LIN {X 50.071,Y -41.479,Z -55.435,A -90.000,B 90.000,C 0.000} C_DIS
LIN {X 50.212,Y -41.479,Z -55.447,A -90.000,B 90.000,C 0.000} C_DIS
LIN {X 50.447,Y -41.466,Z -55.476,A -90.000,B 90.000,C 0.000} C_DIS
LIN {X 50.555,Y -41.461,Z -55.492,A -90.000,B 90.000,C 0.000} C_DIS
LIN {X 50.778,Y -41.444,Z -55.543,A -90.000,B 90.000,C 0.000} C_DIS
LIN {X 51.194,Y -41.423,Z -55.655,A -90.000,B 90.000,C 0.000} C_DIS
LIN {X 51.382,Y -41.418,Z -55.709,A -90.000,B 90.000,C 0.000} C_DIS
LIN {X 51.626,Y -41.420,Z -55.793,A -90.000,B 90.000,C 0.000} C_DIS
LIN {X 51.729,Y -41.422,Z -55.832,A -90.000,B 90.000,C 0.000} C_DIS
LIN {X 52.257,Y -41.443,Z -56.046,A -90.000,B 90.000,C 0.000} C_DIS
LIN {X 52.585,Y -41.450,Z -56.183,A -90.000,B 90.000,C 0.000} C_DIS
LIN {X 52.911,Y -41.433,Z -56.335,A -90.000,B 90.000,C 0.000} C_DIS
LIN {X 53.221,Y -41.399,Z -56.488,A -90.000,B 90.000,C 0.000} C_DIS
LIN {X 53.268,Y -41.394,Z -56.511,A -90.000,B 90.000,C 0.000} C_DIS
LIN {X 53.605,Y -41.331,Z -56.691,A -90.000,B 90.000,C 0.000} C_DIS
LIN {X 53.739,Y -41.308,Z -56.767,A -90.000,B 90.000,C 0.000} C_DIS
LIN {X 53.739,Y -60.000,Z -56.767,A -90.000,B 90.000,C 0.000} C_DIS
LIN {X 39.737,Y -60.000,Z -87.967,A -90.000,B 90.000,C 0.000} C_DIS
LIN {X 39.737,Y -42.859,Z -87.967,A -90.000,B 90.000,C 0.000} C_DIS
LIN {X 40.701,Y -42.857,Z -88.423,A -90.000,B 90.000,C 0.000} C_DIS
LIN {X 40.775,Y -42.860,Z -88.457,A -90.000,B 90.000,C 0.000} C_DIS
LIN {X 41.091,Y -42.861,Z -88.606,A -90.000,B 90.000,C 0.000} C_DIS
LIN {X 41.387,Y -42.856,Z -88.749,A -90.000,B 90.000,C 0.000} C_DIS
LIN {X 41.518,Y -42.856,Z -88.821,A -90.000,B 90.000,C 0.000} C_DIS
LIN {X 41.830,Y -42.856,Z -88.996,A -90.000,B 90.000,C 0.000} C_DIS
LIN {X 41.925,Y -42.857,Z -89.053,A -90.000,B 90.000,C 0.000} C_DIS
LIN {X 42.012,Y -42.859,Z -89.111,A -90.000,B 90.000,C 0.000} C_DIS
LIN {X 42.238,Y -42.866,Z -89.272,A -90.000,B 90.000,C 0.000} C_DIS
LIN {X 42.392,Y -42.871,Z -89.385,A -90.000,B 90.000,C 0.000} C_DIS
LIN {X 42.668,Y -42.871,Z -89.540,A -90.000,B 90.000,C 0.000} C_DIS
LIN {X 43.663,Y -42.840,Z -90.105,A -90.000,B 90.000,C 0.000} C_DIS
LIN {X 43.846,Y -42.837,Z -90.222,A -90.000,B 90.000,C 0.000} C_DIS
LIN {X 44.056,Y -42.836,Z -90.373,A -90.000,B 90.000,C 0.000} C_DIS
LIN {X 44.494,Y -42.834,Z -90.695,A -90.000,B 90.000,C 0.000} C_DIS
LIN {X 44.650,Y -42.831,Z -90.811,A -90.000,B 90.000,C 0.000} C_DIS
LIN {X 44.974,Y -42.816,Z -91.054,A -90.000,B 90.000,C 0.000} C_DIS
LIN {X 45.094,Y -42.815,Z -91.149,A -90.000,B 90.000,C 0.000} C_DIS
LIN {X 45.874,Y -42.815,Z -91.799,A -90.000,B 90.000,C 0.000} C_DIS
LIN {X 45.991,Y -42.817,Z -91.906,A -90.000,B 90.000,C 0.000} C_DIS
LIN {X 46.076,Y -42.820,Z -91.995,A -90.000,B 90.000,C 0.000} C_DIS
LIN {X 46.259,Y -42.829,Z -92.193,A -90.000,B 90.000,C 0.000} C_DIS
LIN {X 46.966,Y -42.829,Z -92.975,A -90.000,B 90.000,C 0.000} C_DIS
LIN {X 47.383,Y -42.820,Z -93.379,A -90.000,B 90.000,C 0.000} C_DIS
LIN {X 47.478,Y -42.813,Z -93.473,A -90.000,B 90.000,C 0.000} C_DIS
LIN {X 47.567,Y -42.807,Z -93.567,A -90.000,B 90.000,C 0.000} C_DIS
LIN {X 47.724,Y -42.799,Z -93.743,A -90.000,B 90.000,C 0.000} C_DIS
LIN {X 47.806,Y -42.796,Z -93.841,A -90.000,B 90.000,C 0.000} C_DIS
LIN {X 48.188,Y -42.784,Z -94.326,A -90.000,B 90.000,C 0.000} C_DIS
LIN {X 48.342,Y -42.784,Z -94.551,A -90.000,B 90.000,C 0.000} C_DIS
LIN {X 48.557,Y -42.792,Z -94.920,A -90.000,B 90.000,C 0.000} C_DIS
LIN {X 49.731,Y -42.798,Z -96.974,A -90.000,B 90.000,C 0.000} C_DIS
LIN {X 50.005,Y -42.776,Z -97.466,A -90.000,B 90.000,C 0.000} C_DIS
LIN {X 50.218,Y -42.754,Z -97.852,A -90.000,B 90.000,C 0.000} C_DIS
LIN {X 50.313,Y -42.746,Z -98.046,A -90.000,B 90.000,C 0.000} C_DIS
LIN {X 50.630,Y -42.732,Z -98.793,A -90.000,B 90.000,C 0.000} C_DIS
LIN {X 50.685,Y -42.731,Z -98.940,A -90.000,B 90.000,C 0.000} C_DIS
LIN {X 50.789,Y -42.732,Z -99.247,A -90.000,B 90.000,C 0.000} C_DIS
LIN {X 50.909,Y -42.728,Z -99.606,A -90.000,B 90.000,C 0.000} C_DIS
LIN {X 50.940,Y -42.728,Z -99.713,A -90.000,B 90.000,C 0.000} C_DIS
LIN {X 51.021,Y -42.724,Z -100.019,A -90.000,B 90.000,C 0.000} C_DIS
LIN {X 51.404,Y -42.715,Z -101.622,A -90.000,B 90.000,C 0.000} C_DIS
LIN {X 51.588,Y -42.705,Z -102.400,A -90.000,B 90.000,C 0.000} C_DIS
LIN {X 51.623,Y -42.698,Z -102.554,A -90.000,B 90.000,C 0.000} C_DIS
LIN {X 51.666,Y -42.691,Z -102.832,A -90.000,B 90.000,C 0.000} C_DIS
LIN {X 51.762,Y -42.691,Z -103.918,A -90.000,B 90.000,C 0.000} C_DIS
LIN {X 51.950,Y -42.585,Z -106.453,A -90.000,B 90.000,C 0.000} C_DIS
LIN {X 51.961,Y -42.579,Z -106.611,A -90.000,B 90.000,C 0.000} C_DIS
LIN {X 51.967,Y -42.576,Z -106.795,A -90.000,B 90.000,C 0.000} C_DIS
LIN {X 51.961,Y -42.576,Z -107.317,A -90.000,B 90.000,C 0.000} C_DIS
LIN {X 51.957,Y -42.578,Z -107.444,A -90.000,B 90.000,C 0.000} C_DIS
LIN {X 51.942,Y -42.583,Z -107.626,A -90.000,B 90.000,C 0.000} C_DIS
LIN {X 51.893,Y -42.599,Z -108.028,A -90.000,B 90.000,C 0.000} C_DIS
LIN {X 51.693,Y -42.585,Z -109.737,A -90.000,B 90.000,C 0.000} C_DIS
LIN {X 51.495,Y -42.558,Z -111.384,A -90.000,B 90.000,C 0.000} C_DIS
LIN {X 51.480,Y -42.556,Z -111.487,A -90.000,B 90.000,C 0.000} C_DIS
LIN {X 51.431,Y -42.553,Z -111.764,A -90.000,B 90.000,C 0.000} C_DIS
LIN {X 51.407,Y -42.554,Z -111.885,A -90.000,B 90.000,C 0.000} C_DIS
LIN {X 51.390,Y -42.555,Z -111.958,A -90.000,B 90.000,C 0.000} C_DIS
LIN {X 51.314,Y -42.552,Z -112.270,A -90.000,B 90.000,C 0.000} C_DIS
LIN {X 51.191,Y -42.541,Z -112.760,A -90.000,B 90.000,C 0.000} C_DIS
LIN {X 50.692,Y -42.505,Z -114.766,A -90.000,B 90.000,C 0.000} C_DIS
LIN {X 50.498,Y -42.486,Z -115.589,A -90.000,B 90.000,C 0.000} C_DIS
LIN {X 50.434,Y -42.486,Z -115.809,A -90.000,B 90.000,C 0.000} C_DIS
LIN {X 50.344,Y -42.494,Z -116.069,A -90.000,B 90.000,C 0.000} C_DIS
LIN {X 49.479,Y -42.446,Z -118.357,A -90.000,B 90.000,C 0.000} C_DIS
LIN {X 49.172,Y -42.430,Z -119.163,A -90.000,B 90.000,C 0.000} C_DIS
LIN {X 49.034,Y -42.425,Z -119.529,A -90.000,B 90.000,C 0.000} C_DIS
LIN {X 48.992,Y -42.424,Z -119.632,A -90.000,B 90.000,C 0.000} C_DIS
LIN {X 48.884,Y -42.426,Z -119.879,A -90.000,B 90.000,C 0.000} C_DIS
LIN {X 48.823,Y -42.428,Z -120.005,A -90.000,B 90.000,C 0.000} C_DIS
LIN {X 48.791,Y -42.431,Z -120.066,A -90.000,B 90.000,C 0.000} C_DIS
LIN {X 48.534,Y -42.422,Z -120.533,A -90.000,B 90.000,C 0.000} C_DIS
LIN {X 47.898,Y -42.413,Z -121.632,A -90.000,B 90.000,C 0.000} C_DIS
LIN {X 46.862,Y -42.389,Z -123.413,A -90.000,B 90.000,C 0.000} C_DIS
LIN {X 46.662,Y -42.391,Z -123.729,A -90.000,B 90.000,C 0.000} C_DIS
LIN {X 46.658,Y -42.391,Z -123.735,A -90.000,B 90.000,C 0.000} C_DIS
LIN {X 46.583,Y -42.387,Z -123.842,A -90.000,B 90.000,C 0.000} C_DIS
LIN {X 46.538,Y -42.386,Z -123.901,A -90.000,B 90.000,C 0.000} C_DIS
LIN {X 46.281,Y -42.383,Z -124.220,A -90.000,B 90.000,C 0.000} C_DIS
LIN {X 44.705,Y -42.346,Z -126.159,A -90.000,B 90.000,C 0.000} C_DIS
LIN {X 43.973,Y -42.339,Z -127.027,A -90.000,B 90.000,C 0.000} C_DIS
LIN {X 43.899,Y -42.333,Z -127.109,A -90.000,B 90.000,C 0.000} C_DIS
LIN {X 43.803,Y -42.329,Z -127.209,A -90.000,B 90.000,C 0.000} C_DIS
LIN {X 41.107,Y -42.265,Z -129.839,A -90.000,B 90.000,C 0.000} C_DIS
LIN {X 40.894,Y -42.262,Z -130.041,A -90.000,B 90.000,C 0.000} C_DIS
LIN {X 40.681,Y -42.253,Z -130.229,A -90.000,B 90.000,C 0.000} C_DIS
LIN {X 38.963,Y -42.211,Z -131.679,A -90.000,B 90.000,C 0.000} C_DIS
LIN {X 37.727,Y -42.184,Z -132.716,A -90.000,B 90.000,C 0.000} C_DIS
LIN {X 37.616,Y -42.182,Z -132.810,A -90.000,B 90.000,C 0.000} C_DIS
LIN {X 37.039,Y -42.183,Z -133.273,A -90.000,B 90.000,C 0.000} C_DIS
LIN {X 34.620,Y -42.128,Z -135.162,A -90.000,B 90.000,C 0.000} C_DIS
LIN {X 33.077,Y -42.091,Z -136.358,A -90.000,B 90.000,C 0.000} C_DIS
LIN {X 32.369,Y -42.096,Z -136.929,A -90.000,B 90.000,C 0.000} C_DIS
LIN {X 31.860,Y -42.079,Z -137.367,A -90.000,B 90.000,C 0.000} C_DIS
LIN {X 31.762,Y -42.078,Z -137.447,A -90.000,B 90.000,C 0.000} C_DIS
LIN {X 30.790,Y -42.057,Z -138.156,A -90.000,B 90.000,C 0.000} C_DIS
LIN {X 30.113,Y -42.060,Z -138.669,A -90.000,B 90.000,C 0.000} C_DIS
LIN {X 28.963,Y -42.027,Z -139.590,A -90.000,B 90.000,C 0.000} C_DIS
LIN {X 28.847,Y -42.027,Z -139.678,A -90.000,B 90.000,C 0.000} C_DIS
LIN {X 28.513,Y -42.013,Z -139.905,A -90.000,B 90.000,C 0.000} C_DIS
LIN {X 27.881,Y -42.005,Z -140.313,A -90.000,B 90.000,C 0.000} C_DIS
LIN {X 26.764,Y -42.006,Z -141.053,A -90.000,B 90.000,C 0.000} C_DIS
LIN {X 25.701,Y -41.985,Z -141.782,A -90.000,B 90.000,C 0.000} C_DIS
LIN {X 25.467,Y -41.978,Z -141.937,A -90.000,B 90.000,C 0.000} C_DIS
LIN {X 25.363,Y -41.981,Z -141.999,A -90.000,B 90.000,C 0.000} C_DIS
LIN {X 25.194,Y -41.978,Z -142.091,A -90.000,B 90.000,C 0.000} C_DIS
LIN {X 23.934,Y -41.975,Z -142.754,A -90.000,B 90.000,C 0.000} C_DIS
LIN {X 22.011,Y -41.953,Z -143.779,A -90.000,B 90.000,C 0.000} C_DIS
LIN {X 21.928,Y -41.954,Z -143.821,A -90.000,B 90.000,C 0.000} C_DIS
LIN {X 21.714,Y -41.959,Z -143.926,A -90.000,B 90.000,C 0.000} C_DIS
LIN {X 21.480,Y -41.961,Z -144.033,A -90.000,B 90.000,C 0.000} C_DIS
LIN {X 21.348,Y -41.966,Z -144.089,A -90.000,B 90.000,C 0.000} C_DIS
LIN {X 18.681,Y -41.946,Z -145.072,A -90.000,B 90.000,C 0.000} C_DIS
LIN {X 17.616,Y -41.939,Z -145.462,A -90.000,B 90.000,C 0.000} C_DIS
LIN {X 17.283,Y -41.941,Z -145.580,A -90.000,B 90.000,C 0.000} C_DIS
LIN {X 16.866,Y -41.961,Z -145.707,A -90.000,B 90.000,C 0.000} C_DIS
LIN {X 16.487,Y -41.974,Z -145.816,A -90.000,B 90.000,C 0.000} C_DIS
LIN {X 14.194,Y -41.972,Z -146.399,A -90.000,B 90.000,C 0.000} C_DIS
LIN {X 12.844,Y -41.974,Z -146.734,A -90.000,B 90.000,C 0.000} C_DIS
LIN {X 12.500,Y -41.983,Z -146.811,A -90.000,B 90.000,C 0.000} C_DIS
LIN {X 12.199,Y -41.993,Z -146.875,A -90.000,B 90.000,C 0.000} C_DIS
LIN {X 11.749,Y -42.015,Z -146.962,A -90.000,B 90.000,C 0.000} C_DIS
LIN {X 11.360,Y -42.023,Z -147.028,A -90.000,B 90.000,C 0.000} C_DIS
LIN {X 9.505,Y -42.021,Z -147.309,A -90.000,B 90.000,C 0.000} C_DIS
LIN {X 7.684,Y -42.033,Z -147.572,A -90.000,B 90.000,C 0.000} C_DIS
LIN {X 7.309,Y -42.042,Z -147.618,A -90.000,B 90.000,C 0.000} C_DIS
LIN {X 7.166,Y -42.049,Z -147.632,A -90.000,B 90.000,C 0.000} C_DIS
LIN {X 6.691,Y -42.078,Z -147.670,A -90.000,B 90.000,C 0.000} C_DIS
LIN {X 6.323,Y -42.091,Z -147.692,A -90.000,B 90.000,C 0.000} C_DIS
LIN {X 5.823,Y -42.090,Z -147.707,A -90.000,B 90.000,C 0.000} C_DIS
LIN {X 3.623,Y -42.092,Z -147.779,A -90.000,B 90.000,C 0.000} C_DIS
LIN {X 3.188,Y -42.091,Z -147.792,A -90.000,B 90.000,C 0.000} C_DIS
LIN {X 2.793,Y -42.094,Z -147.798,A -90.000,B 90.000,C 0.000} C_DIS
LIN {X 2.443,Y -42.104,Z -147.796,A -90.000,B 90.000,C 0.000} C_DIS
LIN {X 2.302,Y -42.111,Z -147.791,A -90.000,B 90.000,C 0.000} C_DIS
LIN {X 2.162,Y -42.121,Z -147.784,A -90.000,B 90.000,C 0.000} C_DIS
LIN {X 1.780,Y -42.138,Z -147.750,A -90.000,B 90.000,C 0.000} C_DIS
LIN {X -1.809,Y -42.140,Z -147.310,A -90.000,B 90.000,C 0.000} C_DIS
LIN {X -2.153,Y -42.146,Z -147.257,A -90.000,B 90.000,C 0.000} C_DIS
LIN {X -2.321,Y -42.149,Z -147.226,A -90.000,B 90.000,C 0.000} C_DIS
LIN {X -2.512,Y -42.161,Z -147.180,A -90.000,B 90.000,C 0.000} C_DIS
LIN {X -5.904,Y -42.185,Z -146.217,A -90.000,B 90.000,C 0.000} C_DIS
LIN {X -6.299,Y -42.185,Z -146.107,A -90.000,B 90.000,C 0.000} C_DIS
LIN {X -6.474,Y -42.187,Z -146.050,A -90.000,B 90.000,C 0.000} C_DIS
LIN {X -6.619,Y -42.192,Z -145.996,A -90.000,B 90.000,C 0.000} C_DIS
LIN {X -6.797,Y -42.187,Z -145.923,A -90.000,B 90.000,C 0.000} C_DIS
LIN {X -6.898,Y -42.187,Z -145.879,A -90.000,B 90.000,C 0.000} C_DIS
LIN {X -9.013,Y -42.202,Z -144.902,A -90.000,B 90.000,C 0.000} C_DIS
LIN {X -10.307,Y -42.229,Z -144.277,A -90.000,B 90.000,C 0.000} C_DIS
LIN {X -10.392,Y -42.227,Z -144.233,A -90.000,B 90.000,C 0.000} C_DIS
LIN {X -10.641,Y -42.224,Z -144.092,A -90.000,B 90.000,C 0.000} C_DIS
LIN {X -10.832,Y -42.222,Z -143.972,A -90.000,B 90.000,C 0.000} C_DIS
LIN {X -10.913,Y -42.223,Z -143.918,A -90.000,B 90.000,C 0.000} C_DIS
LIN {X -11.965,Y -42.251,Z -143.181,A -90.000,B 90.000,C 0.000} C_DIS
LIN {X -13.757,Y -42.332,Z -141.862,A -90.000,B 90.000,C 0.000} C_DIS
LIN {X -13.967,Y -42.332,Z -141.700,A -90.000,B 90.000,C 0.000} C_DIS
LIN {X -14.058,Y -42.333,Z -141.626,A -90.000,B 90.000,C 0.000} C_DIS
LIN {X -14.298,Y -42.335,Z -141.415,A -90.000,B 90.000,C 0.000} C_DIS
LIN {X -14.414,Y -42.339,Z -141.307,A -90.000,B 90.000,C 0.000} C_DIS
LIN {X -14.878,Y -42.372,Z -140.841,A -90.000,B 90.000,C 0.000} C_DIS
LIN {X -15.587,Y -42.405,Z -140.116,A -90.000,B 90.000,C 0.000} C_DIS
LIN {X -15.666,Y -42.411,Z -140.030,A -90.000,B 90.000,C 0.000} C_DIS
LIN {X -15.913,Y -42.435,Z -139.750,A -90.000,B 90.000,C 0.000} C_DIS
LIN {X -16.705,Y -42.506,Z -138.786,A -90.000,B 90.000,C 0.000} C_DIS
LIN {X -16.907,Y -42.509,Z -138.529,A -90.000,B 90.000,C 0.000} C_DIS
LIN {X -17.090,Y -42.502,Z -138.288,A -90.000,B 90.000,C 0.000} C_DIS
LIN {X -17.149,Y -42.500,Z -138.207,A -90.000,B 90.000,C 0.000} C_DIS
LIN {X -17.273,Y -42.500,Z -138.024,A -90.000,B 90.000,C 0.000} C_DIS
LIN {X -17.333,Y -42.502,Z -137.930,A -90.000,B 90.000,C 0.000} C_DIS
LIN {X -17.523,Y -42.510,Z -137.616,A -90.000,B 90.000,C 0.000} C_DIS
LIN {X -17.548,Y -42.512,Z -137.572,A -90.000,B 90.000,C 0.000} C_DIS
LIN {X -18.006,Y -42.548,Z -136.749,A -90.000,B 90.000,C 0.000} C_DIS
LIN {X -18.152,Y -42.554,Z -136.476,A -90.000,B 90.000,C 0.000} C_DIS
LIN {X -18.227,Y -42.560,Z -136.309,A -90.000,B 90.000,C 0.000} C_DIS
LIN {X -18.660,Y -42.596,Z -135.308,A -90.000,B 90.000,C 0.000} C_DIS
LIN {X -18.715,Y -42.603,Z -135.169,A -90.000,B 90.000,C 0.000} C_DIS
LIN {X -18.808,Y -42.619,Z -134.900,A -90.000,B 90.000,C 0.000} C_DIS
LIN {X -18.853,Y -42.629,Z -134.752,A -90.000,B 90.000,C 0.000} C_DIS
LIN {X -18.945,Y -42.658,Z -134.411,A -90.000,B 90.000,C 0.000} C_DIS
LIN {X -19.082,Y -42.685,Z -133.875,A -90.000,B 90.000,C 0.000} C_DIS
LIN {X -19.107,Y -42.689,Z -133.784,A -90.000,B 90.000,C 0.000} C_DIS
LIN {X -19.176,Y -42.693,Z -133.531,A -90.000,B 90.000,C 0.000} C_DIS
LIN {X -19.325,Y -42.693,Z -132.968,A -90.000,B 90.000,C 0.000} C_DIS
LIN {X -19.362,Y -42.695,Z -132.798,A -90.000,B 90.000,C 0.000} C_DIS
LIN {X -19.437,Y -42.713,Z -132.299,A -90.000,B 90.000,C 0.000} C_DIS
LIN {X -19.552,Y -42.713,Z -131.461,A -90.000,B 90.000,C 0.000} C_DIS
LIN {X -19.581,Y -42.717,Z -131.156,A -90.000,B 90.000,C 0.000} C_DIS
LIN {X -19.603,Y -42.724,Z -130.934,A -90.000,B 90.000,C 0.000} C_DIS
LIN {X -19.640,Y -42.751,Z -130.280,A -90.000,B 90.000,C 0.000} C_DIS
LIN {X -19.639,Y -42.759,Z -130.130,A -90.000,B 90.000,C 0.000} C_DIS
LIN {X -19.617,Y -42.789,Z -129.641,A -90.000,B 90.000,C 0.000} C_DIS
LIN {X -19.636,Y -42.801,Z -129.252,A -90.000,B 90.000,C 0.000} C_DIS
LIN {X -19.641,Y -42.803,Z -129.145,A -90.000,B 90.000,C 0.000} C_DIS
LIN {X -19.677,Y -42.803,Z -128.287,A -90.000,B 90.000,C 0.000} C_DIS
LIN {X -19.697,Y -42.805,Z -127.046,A -90.000,B 90.000,C 0.000} C_DIS
LIN {X -19.693,Y -42.809,Z -126.940,A -90.000,B 90.000,C 0.000} C_DIS
LIN {X -19.653,Y -42.844,Z -126.286,A -90.000,B 90.000,C 0.000} C_DIS
LIN {X -19.642,Y -42.858,Z -126.087,A -90.000,B 90.000,C 0.000} C_DIS
LIN {X -19.631,Y -42.879,Z -125.771,A -90.000,B 90.000,C 0.000} C_DIS
LIN {X -19.603,Y -42.899,Z -125.166,A -90.000,B 90.000,C 0.000} C_DIS
LIN {X -19.661,Y -42.899,Z -124.644,A -90.000,B 90.000,C 0.000} C_DIS
LIN {X -19.758,Y -42.891,Z -124.156,A -90.000,B 90.000,C 0.000} C_DIS
LIN {X -19.801,Y -42.891,Z -123.940,A -90.000,B 90.000,C 0.000} C_DIS
LIN {X -20.115,Y -42.903,Z -122.129,A -90.000,B 90.000,C 0.000} C_DIS
LIN {X -20.237,Y -42.923,Z -121.450,A -90.000,B 90.000,C 0.000} C_DIS
LIN {X -20.376,Y -42.942,Z -120.661,A -90.000,B 90.000,C 0.000} C_DIS
LIN {X -20.581,Y -42.942,Z -119.994,A -90.000,B 90.000,C 0.000} C_DIS
LIN {X -21.455,Y -42.935,Z -117.314,A -90.000,B 90.000,C 0.000} C_DIS
LIN {X -21.829,Y -42.941,Z -116.105,A -90.000,B 90.000,C 0.000} C_DIS
LIN {X -22.072,Y -42.942,Z -115.374,A -90.000,B 90.000,C 0.000} C_DIS
LIN {X -22.994,Y -42.949,Z -112.548,A -90.000,B 90.000,C 0.000} C_DIS
LIN {X -23.502,Y -42.948,Z -111.018,A -90.000,B 90.000,C 0.000} C_DIS
LIN {X -23.968,Y -42.918,Z -109.597,A -90.000,B 90.000,C 0.000} C_DIS
LIN {X -23.994,Y -42.917,Z -109.512,A -90.000,B 90.000,C 0.000} C_DIS
LIN {X -24.144,Y -42.910,Z -108.976,A -90.000,B 90.000,C 0.000} C_DIS
LIN {X -24.171,Y -42.910,Z -108.866,A -90.000,B 90.000,C 0.000} C_DIS
LIN {X -24.570,Y -42.910,Z -107.060,A -90.000,B 90.000,C 0.000} C_DIS
LIN {X -24.799,Y -42.909,Z -106.089,A -90.000,B 90.000,C 0.000} C_DIS
LIN {X -24.962,Y -42.917,Z -105.256,A -90.000,B 90.000,C 0.000} C_DIS
LIN {X -25.003,Y -42.913,Z -105.043,A -90.000,B 90.000,C 0.000} C_DIS
LIN {X -25.151,Y -42.884,Z -104.254,A -90.000,B 90.000,C 0.000} C_DIS
LIN {X -25.364,Y -42.835,Z -103.100,A -90.000,B 90.000,C 0.000} C_DIS
LIN {X -25.393,Y -42.828,Z -102.931,A -90.000,B 90.000,C 0.000} C_DIS
LIN {X -25.429,Y -42.820,Z -102.650,A -90.000,B 90.000,C 0.000} C_DIS
LIN {X -25.473,Y -42.813,Z -102.168,A -90.000,B 90.000,C 0.000} C_DIS
LIN {X -25.479,Y -42.813,Z -102.068,A -90.000,B 90.000,C 0.000} C_DIS
LIN {X -25.481,Y -42.813,Z -101.989,A -90.000,B 90.000,C 0.000} C_DIS
LIN {X -25.478,Y -42.815,Z -101.889,A -90.000,B 90.000,C 0.000} C_DIS
LIN {X -25.459,Y -42.823,Z -101.480,A -90.000,B 90.000,C 0.000} C_DIS
LIN {X -25.418,Y -42.823,Z -100.675,A -90.000,B 90.000,C 0.000} C_DIS
LIN {X -25.361,Y -42.824,Z -99.605,A -90.000,B 90.000,C 0.000} C_DIS
LIN {X -25.342,Y -42.826,Z -99.369,A -90.000,B 90.000,C 0.000} C_DIS
LIN {X -25.324,Y -42.828,Z -99.221,A -90.000,B 90.000,C 0.000} C_DIS
LIN {X -25.232,Y -42.841,Z -98.696,A -90.000,B 90.000,C 0.000} C_DIS
LIN {X -25.060,Y -42.822,Z -97.787,A -90.000,B 90.000,C 0.000} C_DIS
LIN {X -24.931,Y -42.812,Z -97.157,A -90.000,B 90.000,C 0.000} C_DIS
LIN {X -24.835,Y -42.801,Z -96.697,A -90.000,B 90.000,C 0.000} C_DIS
LIN {X -24.789,Y -42.800,Z -96.516,A -90.000,B 90.000,C 0.000} C_DIS
LIN {X -24.691,Y -42.803,Z -96.198,A -90.000,B 90.000,C 0.000} C_DIS
LIN {X -24.588,Y -42.801,Z -95.935,A -90.000,B 90.000,C 0.000} C_DIS
LIN {X -24.293,Y -42.788,Z -95.204,A -90.000,B 90.000,C 0.000} C_DIS
LIN {X -23.710,Y -42.779,Z -93.880,A -90.000,B 90.000,C 0.000} C_DIS
LIN {X -23.646,Y -42.780,Z -93.748,A -90.000,B 90.000,C 0.000} C_DIS
LIN {X -23.509,Y -42.774,Z -93.503,A -90.000,B 90.000,C 0.000} C_DIS
LIN {X -23.438,Y -42.772,Z -93.387,A -90.000,B 90.000,C 0.000} C_DIS
LIN {X -22.930,Y -42.770,Z -92.617,A -90.000,B 90.000,C 0.000} C_DIS
LIN {X -22.141,Y -42.778,Z -91.478,A -90.000,B 90.000,C 0.000} C_DIS
LIN {X -22.025,Y -42.771,Z -91.315,A -90.000,B 90.000,C 0.000} C_DIS
LIN {X -21.895,Y -42.767,Z -91.150,A -90.000,B 90.000,C 0.000} C_DIS
LIN {X -21.739,Y -42.767,Z -90.971,A -90.000,B 90.000,C 0.000} C_DIS
LIN {X -21.638,Y -42.768,Z -90.861,A -90.000,B 90.000,C 0.000} C_DIS
LIN {X -20.770,Y -42.781,Z -89.942,A -90.000,B 90.000,C 0.000} C_DIS
LIN {X -20.233,Y -42.786,Z -89.381,A -90.000,B 90.000,C 0.000} C_DIS
LIN {X -19.786,Y -42.770,Z -88.923,A -90.000,B 90.000,C 0.000} C_DIS
LIN {X -19.740,Y -42.769,Z -88.881,A -90.000,B 90.000,C 0.000} C_DIS
LIN {X -19.644,Y -42.769,Z -88.799,A -90.000,B 90.000,C 0.000} C_DIS
LIN {X -18.038,Y -42.776,Z -87.523,A -90.000,B 90.000,C 0.000} C_DIS
LIN {X -17.889,Y -42.774,Z -87.405,A -90.000,B 90.000,C 0.000} C_DIS
LIN {X -17.261,Y -42.760,Z -86.913,A -90.000,B 90.000,C 0.000} C_DIS
LIN {X -17.070,Y -42.757,Z -86.771,A -90.000,B 90.000,C 0.000} C_DIS
LIN {X -16.961,Y -42.757,Z -86.694,A -90.000,B 90.000,C 0.000} C_DIS
LIN {X -16.811,Y -42.759,Z -86.600,A -90.000,B 90.000,C 0.000} C_DIS
LIN {X -16.710,Y -42.761,Z -86.541,A -90.000,B 90.000,C 0.000} C_DIS
LIN {X -16.482,Y -42.769,Z -86.418,A -90.000,B 90.000,C 0.000} C_DIS
LIN {X -14.960,Y -42.789,Z -85.602,A -90.000,B 90.000,C 0.000} C_DIS
LIN {X -14.663,Y -42.786,Z -85.445,A -90.000,B 90.000,C 0.000} C_DIS
LIN {X -14.565,Y -42.786,Z -85.396,A -90.000,B 90.000,C 0.000} C_DIS
LIN {X -14.302,Y -42.786,Z -85.276,A -90.000,B 90.000,C 0.000} C_DIS
LIN {X -13.760,Y -42.781,Z -85.045,A -90.000,B 90.000,C 0.000} C_DIS
LIN {X -13.186,Y -42.770,Z -84.803,A -90.000,B 90.000,C 0.000} C_DIS
LIN {X -13.060,Y -42.768,Z -84.754,A -90.000,B 90.000,C 0.000} C_DIS
LIN {X -12.089,Y -42.768,Z -84.417,A -90.000,B 90.000,C 0.000} C_DIS
LIN {X -11.927,Y -42.763,Z -84.363,A -90.000,B 90.000,C 0.000} C_DIS
LIN {X -11.822,Y -42.760,Z -84.330,A -90.000,B 90.000,C 0.000} C_DIS
LIN {X -11.726,Y -42.760,Z -84.306,A -90.000,B 90.000,C 0.000} C_DIS
LIN {X -10.567,Y -42.760,Z -84.040,A -90.000,B 90.000,C 0.000} C_DIS
LIN {X -10.058,Y -42.756,Z -83.924,A -90.000,B 90.000,C 0.000} C_DIS
LIN {X -9.466,Y -42.746,Z -83.796,A -90.000,B 90.000,C 0.000} C_DIS
LIN {X -9.197,Y -42.738,Z -83.739,A -90.000,B 90.000,C 0.000} C_DIS
LIN {X -8.994,Y -42.729,Z -83.697,A -90.000,B 90.000,C 0.000} C_DIS
LIN {X -8.798,Y -42.723,Z -83.666,A -90.000,B 90.000,C 0.000} C_DIS
LIN {X -7.721,Y -42.707,Z -83.549,A -90.000,B 90.000,C 0.000} C_DIS
LIN {X -6.726,Y -42.697,Z -83.455,A -90.000,B 90.000,C 0.000} C_DIS
LIN {X -6.520,Y -42.697,Z -83.442,A -90.000,B 90.000,C 0.000} C_DIS
LIN {X -5.641,Y -42.674,Z -83.394,A -90.000,B 90.000,C 0.000} C_DIS
LIN {X -5.474,Y -42.672,Z -83.391,A -90.000,B 90.000,C 0.000} C_DIS
LIN {X -4.645,Y -42.671,Z -83.411,A -90.000,B 90.000,C 0.000} C_DIS
LIN {X -3.883,Y -42.669,Z -83.422,A -90.000,B 90.000,C 0.000} C_DIS
LIN {X -3.442,Y -42.661,Z -83.431,A -90.000,B 90.000,C 0.000} C_DIS
LIN {X -2.548,Y -42.628,Z -83.454,A -90.000,B 90.000,C 0.000} C_DIS
LIN {X -2.452,Y -42.626,Z -83.459,A -90.000,B 90.000,C 0.000} C_DIS
LIN {X -2.131,Y -42.620,Z -83.482,A -90.000,B 90.000,C 0.000} C_DIS
LIN {X -0.458,Y -42.601,Z -83.632,A -90.000,B 90.000,C 0.000} C_DIS
LIN {X 0.509,Y -42.574,Z -83.726,A -90.000,B 90.000,C 0.000} C_DIS
LIN {X 0.844,Y -42.564,Z -83.754,A -90.000,B 90.000,C 0.000} C_DIS
LIN {X 0.939,Y -42.561,Z -83.764,A -90.000,B 90.000,C 0.000} C_DIS
LIN {X 1.741,Y -42.552,Z -83.868,A -90.000,B 90.000,C 0.000} C_DIS
LIN {X 2.652,Y -42.551,Z -84.004,A -90.000,B 90.000,C 0.000} C_DIS
LIN {X 3.065,Y -42.548,Z -84.067,A -90.000,B 90.000,C 0.000} C_DIS
LIN {X 4.080,Y -42.534,Z -84.225,A -90.000,B 90.000,C 0.000} C_DIS
LIN {X 4.520,Y -42.530,Z -84.299,A -90.000,B 90.000,C 0.000} C_DIS
LIN {X 4.880,Y -42.530,Z -84.367,A -90.000,B 90.000,C 0.000} C_DIS
LIN {X 5.595,Y -42.525,Z -84.487,A -90.000,B 90.000,C 0.000} C_DIS
LIN {X 6.014,Y -42.524,Z -84.557,A -90.000,B 90.000,C 0.000} C_DIS
LIN {X 6.984,Y -42.514,Z -84.721,A -90.000,B 90.000,C 0.000} C_DIS
LIN {X 7.467,Y -42.505,Z -84.805,A -90.000,B 90.000,C 0.000} C_DIS
LIN {X 8.607,Y -42.495,Z -85.028,A -90.000,B 90.000,C 0.000} C_DIS
LIN {X 9.101,Y -42.480,Z -85.117,A -90.000,B 90.000,C 0.000} C_DIS
LIN {X 10.234,Y -42.464,Z -85.313,A -90.000,B 90.000,C 0.000} C_DIS
LIN {X 11.147,Y -42.455,Z -85.480,A -90.000,B 90.000,C 0.000} C_DIS
LIN {X 11.899,Y -42.440,Z -85.622,A -90.000,B 90.000,C 0.000} C_DIS
LIN {X 12.393,Y -42.425,Z -85.705,A -90.000,B 90.000,C 0.000} C_DIS
LIN {X 12.960,Y -42.420,Z -85.795,A -90.000,B 90.000,C 0.000} C_DIS
LIN {X 13.931,Y -42.408,Z -85.945,A -90.000,B 90.000,C 0.000} C_DIS
LIN {X 15.025,Y -42.390,Z -86.117,A -90.000,B 90.000,C 0.000} C_DIS
LIN {X 15.372,Y -42.382,Z -86.166,A -90.000,B 90.000,C 0.000} C_DIS
LIN {X 15.516,Y -42.378,Z -86.183,A -90.000,B 90.000,C 0.000} C_DIS
LIN {X 15.895,Y -42.373,Z -86.226,A -90.000,B 90.000,C 0.000} C_DIS
LIN {X 16.971,Y -42.367,Z -86.345,A -90.000,B 90.000,C 0.000} C_DIS
LIN {X 17.986,Y -42.373,Z -86.482,A -90.000,B 90.000,C 0.000} C_DIS
LIN {X 18.166,Y -42.372,Z -86.503,A -90.000,B 90.000,C 0.000} C_DIS
LIN {X 18.407,Y -42.369,Z -86.528,A -90.000,B 90.000,C 0.000} C_DIS
LIN {X 19.258,Y -42.383,Z -86.601,A -90.000,B 90.000,C 0.000} C_DIS
LIN {X 20.285,Y -42.393,Z -86.693,A -90.000,B 90.000,C 0.000} C_DIS
LIN {X 20.931,Y -42.383,Z -86.723,A -90.000,B 90.000,C 0.000} C_DIS
LIN {X 21.175,Y -42.386,Z -86.732,A -90.000,B 90.000,C 0.000} C_DIS
LIN {X 22.863,Y -42.420,Z -86.825,A -90.000,B 90.000,C 0.000} C_DIS
LIN {X 22.911,Y -42.420,Z -86.825,A -90.000,B 90.000,C 0.000} C_DIS
LIN {X 24.655,Y -42.462,Z -86.776,A -90.000,B 90.000,C 0.000} C_DIS
LIN {X 24.759,Y -42.466,Z -86.775,A -90.000,B 90.000,C 0.000} C_DIS
LIN {X 25.137,Y -42.486,Z -86.788,A -90.000,B 90.000,C 0.000} C_DIS
LIN {X 25.452,Y -42.495,Z -86.773,A -90.000,B 90.000,C 0.000} C_DIS
LIN {X 27.457,Y -42.555,Z -86.702,A -90.000,B 90.000,C 0.000} C_DIS
LIN {X 28.004,Y -42.592,Z -86.675,A -90.000,B 90.000,C 0.000} C_DIS
LIN {X 28.372,Y -42.607,Z -86.627,A -90.000,B 90.000,C 0.000} C_DIS
LIN {X 28.482,Y -42.612,Z -86.615,A -90.000,B 90.000,C 0.000} C_DIS
LIN {X 28.602,Y -42.620,Z -86.610,A -90.000,B 90.000,C 0.000} C_DIS
LIN {X 28.897,Y -42.643,Z -86.605,A -90.000,B 90.000,C 0.000} C_DIS
LIN {X 29.191,Y -42.654,Z -86.604,A -90.000,B 90.000,C 0.000} C_DIS
LIN {X 29.516,Y -42.663,Z -86.604,A -90.000,B 90.000,C 0.000} C_DIS
LIN {X 30.151,Y -42.682,Z -86.604,A -90.000,B 90.000,C 0.000} C_DIS
LIN {X 31.448,Y -42.748,Z -86.597,A -90.000,B 90.000,C 0.000} C_DIS
LIN {X 32.407,Y -42.774,Z -86.504,A -90.000,B 90.000,C 0.000} C_DIS
LIN {X 32.593,Y -42.782,Z -86.498,A -90.000,B 90.000,C 0.000} C_DIS
LIN {X 32.863,Y -42.796,Z -86.495,A -90.000,B 90.000,C 0.000} C_DIS
LIN {X 33.009,Y -42.805,Z -86.501,A -90.000,B 90.000,C 0.000} C_DIS
LIN {X 34.166,Y -42.820,Z -86.560,A -90.000,B 90.000,C 0.000} C_DIS
LIN {X 34.310,Y -42.823,Z -86.572,A -90.000,B 90.000,C 0.000} C_DIS
LIN {X 34.471,Y -42.830,Z -86.599,A -90.000,B 90.000,C 0.000} C_DIS
LIN {X 34.747,Y -42.843,Z -86.652,A -90.000,B 90.000,C 0.000} C_DIS
LIN {X 36.471,Y -42.856,Z -87.005,A -90.000,B 90.000,C 0.000} C_DIS
LIN {X 36.760,Y -42.861,Z -87.044,A -90.000,B 90.000,C 0.000} C_DIS
LIN {X 36.851,Y -42.864,Z -87.060,A -90.000,B 90.000,C 0.000} C_DIS
LIN {X 37.069,Y -42.864,Z -87.105,A -90.000,B 90.000,C 0.000} C_DIS
LIN {X 37.278,Y -42.866,Z -87.156,A -90.000,B 90.000,C 0.000} C_DIS
LIN {X 37.422,Y -42.866,Z -87.198,A -90.000,B 90.000,C 0.000} C_DIS
LIN {X 38.919,Y -42.875,Z -87.668,A -90.000,B 90.000,C 0.000} C_DIS
LIN {X 39.328,Y -42.865,Z -87.799,A -90.000,B 90.000,C 0.000} C_DIS
LIN {X 39.422,Y -42.862,Z -87.832,A -90.000,B 90.000,C 0.000} C_DIS
LIN {X 39.508,Y -42.861,Z -87.866,A -90.000,B 90.000,C 0.000} C_DIS
LIN {X 39.737,Y -42.859,Z -87.967,A -90.000,B 90.000,C 0.000} C_DIS
LIN {X 39.737,Y -60.000,Z -87.967,A -90.000,B 90.000,C 0.000} C_DIS
LIN {X -16.493,Y -60.000,Z -141.596,A -90.000,B 90.000,C 0.000} C_DIS
LIN {X -16.493,Y -41.308,Z -141.596,A -90.000,B 90.000,C 0.000} C_DIS
LIN {X -16.840,Y -41.337,Z -141.251,A -90.000,B 90.000,C 0.000} C_DIS
LIN {X -16.985,Y -41.353,Z -141.099,A -90.000,B 90.000,C 0.000} C_DIS
LIN {X -17.267,Y -41.392,Z -140.789,A -90.000,B 90.000,C 0.000} C_DIS
LIN {X -17.520,Y -41.430,Z -140.496,A -90.000,B 90.000,C 0.000} C_DIS
LIN {X -17.710,Y -41.452,Z -140.270,A -90.000,B 90.000,C 0.000} C_DIS
LIN {X -17.920,Y -41.469,Z -140.012,A -90.000,B 90.000,C 0.000} C_DIS
LIN {X -18.483,Y -41.501,Z -139.316,A -90.000,B 90.000,C 0.000} C_DIS
LIN {X -18.597,Y -41.510,Z -139.168,A -90.000,B 90.000,C 0.000} C_DIS
LIN {X -18.749,Y -41.527,Z -138.958,A -90.000,B 90.000,C 0.000} C_DIS
LIN {X -18.846,Y -41.541,Z -138.818,A -90.000,B 90.000,C 0.000} C_DIS
LIN {X -19.009,Y -41.570,Z -138.571,A -90.000,B 90.000,C 0.000} C_DIS
LIN {X -19.116,Y -41.586,Z -138.400,A -90.000,B 90.000,C 0.000} C_DIS
LIN {X -19.679,Y -41.692,Z -137.451,A -90.000,B 90.000,C 0.000} C_DIS
LIN {X -19.771,Y -41.710,Z -137.293,A -90.000,B 90.000,C 0.000} C_DIS
LIN {X -19.835,Y -41.727,Z -137.173,A -90.000,B 90.000,C 0.000} C_DIS
LIN {X -20.051,Y -41.785,Z -136.725,A -90.000,B 90.000,C 0.000} C_DIS
LIN {X -20.116,Y -41.801,Z -136.586,A -90.000,B 90.000,C 0.000} C_DIS
LIN {X -20.247,Y -41.825,Z -136.298,A -90.000,B 90.000,C 0.000} C_DIS
LIN {X -20.348,Y -41.839,Z -136.070,A -90.000,B 90.000,C 0.000} C_DIS
LIN {X -20.398,Y -41.843,Z -135.951,A -90.000,B 90.000,C 0.000} C_DIS
LIN {X -20.479,Y -41.852,Z -135.739,A -90.000,B 90.000,C 0.000} C_DIS
LIN {X -20.569,Y -41.867,Z -135.477,A -90.000,B 90.000,C 0.000} C_DIS
LIN {X -20.634,Y -41.881,Z -135.272,A -90.000,B 90.000,C 0.000} C_DIS
LIN {X -20.670,Y -41.890,Z -135.146,A -90.000,B 90.000,C 0.000} C_DIS
LIN {X -20.901,Y -41.963,Z -134.286,A -90.000,B 90.000,C 0.000} C_DIS
LIN {X -20.977,Y -41.981,Z -134.030,A -90.000,B 90.000,C 0.000} C_DIS
LIN {X -21.150,Y -42.007,Z -133.412,A -90.000,B 90.000,C 0.000} C_DIS
LIN {X -21.202,Y -42.019,Z -133.195,A -90.000,B 90.000,C 0.000} C_DIS
LIN {X -21.230,Y -42.029,Z -133.055,A -90.000,B 90.000,C 0.000} C_DIS
LIN {X -21.356,Y -42.091,Z -132.295,A -90.000,B 90.000,C 0.000} C_DIS
LIN {X -21.424,Y -42.121,Z -131.871,A -90.000,B 90.000,C 0.000} C_DIS
LIN {X -21.456,Y -42.134,Z -131.653,A -90.000,B 90.000,C 0.000} C_DIS
LIN {X -21.505,Y -42.150,Z -131.159,A -90.000,B 90.000,C 0.000} C_DIS
LIN {X -21.518,Y -42.154,Z -131.016,A -90.000,B 90.000,C 0.000} C_DIS
LIN {X -21.552,Y -42.181,Z -130.414,A -90.000,B 90.000,C 0.000} C_DIS
LIN {X -21.559,Y -42.189,Z -130.235,A -90.000,B 90.000,C 0.000} C_DIS
LIN {X -21.556,Y -42.203,Z -130.009,A -90.000,B 90.000,C 0.000} C_DIS
LIN {X -21.538,Y -42.227,Z -129.621,A -90.000,B 90.000,C 0.000} C_DIS
LIN {X -21.585,Y -42.257,Z -128.709,A -90.000,B 90.000,C 0.000} C_DIS
LIN {X -21.606,Y -42.278,Z -128.317,A -90.000,B 90.000,C 0.000} C_DIS
LIN {X -21.614,Y -42.292,Z -128.080,A -90.000,B 90.000,C 0.000} C_DIS
LIN {X -21.632,Y -42.332,Z -127.593,A -90.000,B 90.000,C 0.000} C_DIS
LIN {X -21.644,Y -42.349,Z -127.058,A -90.000,B 90.000,C 0.000} C_DIS
LIN {X -21.643,Y -42.353,Z -126.957,A -90.000,B 90.000,C 0.000} C_DIS
LIN {X -21.637,Y -42.361,Z -126.799,A -90.000,B 90.000,C 0.000} C_DIS
LIN {X -21.590,Y -42.401,Z -126.030,A -90.000,B 90.000,C 0.000} C_DIS
LIN {X -21.559,Y -42.455,Z -125.223,A -90.000,B 90.000,C 0.000} C_DIS
LIN {X -21.592,Y -42.463,Z -124.946,A -90.000,B 90.000,C 0.000} C_DIS
LIN {X -21.727,Y -42.470,Z -124.273,A -90.000,B 90.000,C 0.000} C_DIS
LIN {X -21.841,Y -42.480,Z -123.624,A -90.000,B 90.000,C 0.000} C_DIS
LIN {X -22.142,Y -42.500,Z -121.903,A -90.000,B 90.000,C 0.000} C_DIS
LIN {X -22.284,Y -42.531,Z -121.117,A -90.000,B 90.000,C 0.000} C_DIS
LIN {X -22.454,Y -42.538,Z -120.569,A -90.000,B 90.000,C 0.000} C_DIS
LIN {X -22.608,Y -42.540,Z -120.101,A -90.000,B 90.000,C 0.000} C_DIS
LIN {X -22.934,Y -42.540,Z -119.102,A -90.000,B 90.000,C 0.000} C_DIS
LIN {X -23.330,Y -42.546,Z -117.893,A -90.000,B 90.000,C 0.000} C_DIS
LIN {X -23.703,Y -42.556,Z -116.689,A -90.000,B 90.000,C 0.000} C_DIS
LIN {X -23.962,Y -42.559,Z -115.910,A -90.000,B 90.000,C 0.000} C_DIS
LIN {X -24.708,Y -42.572,Z -113.627,A -90.000,B 90.000,C 0.000} C_DIS
LIN {X -24.927,Y -42.563,Z -112.955,A -90.000,B 90.000,C 0.000} C_DIS
LIN {X -25.840,Y -42.514,Z -110.172,A -90.000,B 90.000,C 0.000} C_DIS
LIN {X -25.877,Y -42.512,Z -110.051,A -90.000,B 90.000,C 0.000} C_DIS
LIN {X -26.019,Y -42.508,Z -109.544,A -90.000,B 90.000,C 0.000} C_DIS
LIN {X -26.084,Y -42.506,Z -109.288,A -90.000,B 90.000,C 0.000} C_DIS
LIN {X -26.330,Y -42.508,Z -108.174,A -90.000,B 90.000,C 0.000} C_DIS
LIN {X -26.374,Y -42.503,Z -107.969,A -90.000,B 90.000,C 0.000} C_DIS
LIN {X -26.477,Y -42.481,Z -107.481,A -90.000,B 90.000,C 0.000} C_DIS
LIN {X -26.614,Y -42.450,Z -106.873,A -90.000,B 90.000,C 0.000} C_DIS
LIN {X -26.706,Y -42.432,Z -106.458,A -90.000,B 90.000,C 0.000} C_DIS
LIN {X -26.920,Y -42.391,Z -105.300,A -90.000,B 90.000,C 0.000} C_DIS
LIN {X -27.046,Y -42.368,Z -104.628,A -90.000,B 90.000,C 0.000} C_DIS
LIN {X -27.269,Y -42.330,Z -103.443,A -90.000,B 90.000,C 0.000} C_DIS
LIN {X -27.311,Y -42.324,Z -103.190,A -90.000,B 90.000,C 0.000} C_DIS
LIN {X -27.347,Y -42.310,Z -102.900,A -90.000,B 90.000,C 0.000} C_DIS
LIN {X -27.393,Y -42.291,Z -102.366,A -90.000,B 90.000,C 0.000} C_DIS
LIN {X -27.404,Y -42.285,Z -102.193,A -90.000,B 90.000,C 0.000} C_DIS
LIN {X -27.407,Y -42.277,Z -102.024,A -90.000,B 90.000,C 0.000} C_DIS
LIN {X -27.402,Y -42.271,Z -101.835,A -90.000,B 90.000,C 0.000} C_DIS
LIN {X -27.349,Y -42.255,Z -100.894,A -90.000,B 90.000,C 0.000} C_DIS
LIN {X -27.326,Y -42.251,Z -100.478,A -90.000,B 90.000,C 0.000} C_DIS
LIN {X -27.313,Y -42.243,Z -100.269,A -90.000,B 90.000,C 0.000} C_DIS
LIN {X -27.259,Y -42.213,Z -99.443,A -90.000,B 90.000,C 0.000} C_DIS
LIN {X -27.229,Y -42.206,Z -99.134,A -90.000,B 90.000,C 0.000} C_DIS
LIN {X -27.210,Y -42.205,Z -98.987,A -90.000,B 90.000,C 0.000} C_DIS
LIN {X -27.193,Y -42.205,Z -98.877,A -90.000,B 90.000,C 0.000} C_DIS
LIN {X -27.025,Y -42.214,Z -97.939,A -90.000,B 90.000,C 0.000} C_DIS
LIN {X -26.973,Y -42.211,Z -97.659,A -90.000,B 90.000,C 0.000} C_DIS
LIN {X -26.907,Y -42.202,Z -97.325,A -90.000,B 90.000,C 0.000} C_DIS
LIN {X -26.700,Y -42.181,Z -96.325,A -90.000,B 90.000,C 0.000} C_DIS
LIN {X -26.679,Y -42.180,Z -96.233,A -90.000,B 90.000,C 0.000} C_DIS
LIN {X -26.633,Y -42.179,Z -96.052,A -90.000,B 90.000,C 0.000} C_DIS
LIN {X -26.606,Y -42.179,Z -95.956,A -90.000,B 90.000,C 0.000} C_DIS
LIN {X -26.545,Y -42.182,Z -95.756,A -90.000,B 90.000,C 0.000} C_DIS
LIN {X -26.506,Y -42.181,Z -95.631,A -90.000,B 90.000,C 0.000} C_DIS
LIN {X -26.462,Y -42.183,Z -95.504,A -90.000,B 90.000,C 0.000} C_DIS
LIN {X -26.390,Y -42.187,Z -95.317,A -90.000,B 90.000,C 0.000} C_DIS
LIN {X -26.263,Y -42.184,Z -94.999,A -90.000,B 90.000,C 0.000} C_DIS
LIN {X -26.060,Y -42.170,Z -94.502,A -90.000,B 90.000,C 0.000} C_DIS
LIN {X -25.450,Y -42.149,Z -93.120,A -90.000,B 90.000,C 0.000} C_DIS
LIN {X -25.345,Y -42.149,Z -92.901,A -90.000,B 90.000,C 0.000} C_DIS
LIN {X -25.169,Y -42.140,Z -92.585,A -90.000,B 90.000,C 0.000} C_DIS
LIN {X -25.059,Y -42.138,Z -92.402,A -90.000,B 90.000,C 0.000} C_DIS
LIN {X -24.527,Y -42.142,Z -91.589,A -90.000,B 90.000,C 0.000} C_DIS
LIN {X -24.157,Y -42.151,Z -91.051,A -90.000,B 90.000,C 0.000} C_DIS
LIN {X -23.878,Y -42.159,Z -90.645,A -90.000,B 90.000,C 0.000} C_DIS
LIN {X -23.587,Y -42.147,Z -90.233,A -90.000,B 90.000,C 0.000} C_DIS
LIN {X -23.395,Y -42.145,Z -89.982,A -90.000,B 90.000,C 0.000} C_DIS
LIN {X -23.328,Y -42.146,Z -89.901,A -90.000,B 90.000,C 0.000} C_DIS
LIN {X -23.134,Y -42.151,Z -89.676,A -90.000,B 90.000,C 0.000} C_DIS
LIN {X -22.866,Y -42.157,Z -89.389,A -90.000,B 90.000,C 0.000} C_DIS
LIN {X -22.143,Y -42.171,Z -88.622,A -90.000,B 90.000,C 0.000} C_DIS
LIN {X -22.000,Y -42.172,Z -88.473,A -90.000,B 90.000,C 0.000} C_DIS
LIN {X -21.572,Y -42.161,Z -88.032,A -90.000,B 90.000,C 0.000} C_DIS
LIN {X -21.157,Y -42.153,Z -87.604,A -90.000,B 90.000,C 0.000} C_DIS
LIN {X -21.042,Y -42.153,Z -87.493,A -90.000,B 90.000,C 0.000} C_DIS
LIN {X -20.972,Y -42.154,Z -87.430,A -90.000,B 90.000,C 0.000} C_DIS
LIN {X -20.827,Y -42.157,Z -87.307,A -90.000,B 90.000,C 0.000} C_DIS
LIN {X -19.854,Y -42.190,Z -86.522,A -90.000,B 90.000,C 0.000} C_DIS
LIN {X -19.154,Y -42.199,Z -85.964,A -90.000,B 90.000,C 0.000} C_DIS
LIN {X -18.411,Y -42.192,Z -85.378,A -90.000,B 90.000,C 0.000} C_DIS
LIN {X -18.175,Y -42.193,Z -85.202,A -90.000,B 90.000,C 0.000} C_DIS
LIN {X -17.977,Y -42.196,Z -85.065,A -90.000,B 90.000,C 0.000} C_DIS
LIN {X -17.852,Y -42.200,Z -84.986,A -90.000,B 90.000,C 0.000} C_DIS
LIN {X -17.687,Y -42.206,Z -84.887,A -90.000,B 90.000,C 0.000} C_DIS
LIN {X -17.568,Y -42.210,Z -84.820,A -90.000,B 90.000,C 0.000} C_DIS
LIN {X -17.106,Y -42.229,Z -84.568,A -90.000,B 90.000,C 0.000} C_DIS
LIN {X -15.515,Y -42.217,Z -83.727,A -90.000,B 90.000,C 0.000} C_DIS
LIN {X -15.364,Y -42.218,Z -83.653,A -90.000,B 90.000,C 0.000} C_DIS
LIN {X -15.040,Y -42.220,Z -83.505,A -90.000,B 90.000,C 0.000} C_DIS
LIN {X -14.772,Y -42.220,Z -83.390,A -90.000,B 90.000,C 0.000} C_DIS
LIN {X -13.880,Y -42.212,Z -83.012,A -90.000,B 90.000,C 0.000} C_DIS
LIN {X -13.674,Y -42.212,Z -82.934,A -90.000,B 90.000,C 0.000} C_DIS
LIN {X -13.064,Y -42.217,Z -82.721,A -90.000,B 90.000,C 0.000} C_DIS
LIN {X -12.673,Y -42.212,Z -82.586,A -90.000,B 90.000,C 0.000} C_DIS
LIN {X -12.506,Y -42.205,Z -82.531,A -90.000,B 90.000,C 0.000} C_DIS
LIN {X -12.400,Y -42.200,Z -82.499,A -90.000,B 90.000,C 0.000} C_DIS
LIN {X -12.251,Y -42.195,Z -82.459,A -90.000,B 90.000,C 0.000} C_DIS
LIN {X -12.155,Y -42.193,Z -82.436,A -90.000,B 90.000,C 0.000} C_DIS
LIN {X -10.404,Y -42.160,Z -82.045,A -90.000,B 90.000,C 0.000} C_DIS
LIN {X -10.155,Y -42.155,Z -81.992,A -90.000,B 90.000,C 0.000} C_DIS
LIN {X -9.878,Y -42.144,Z -81.934,A -90.000,B 90.000,C 0.000} C_DIS
LIN {X -9.406,Y -42.123,Z -81.836,A -90.000,B 90.000,C 0.000} C_DIS
LIN {X -9.308,Y -42.119,Z -81.818,A -90.000,B 90.000,C 0.000} C_DIS
LIN {X -9.056,Y -42.112,Z -81.780,A -90.000,B 90.000,C 0.000} C_DIS
LIN {X -9.013,Y -42.111,Z -81.774,A -90.000,B 90.000,C 0.000} C_DIS
LIN {X -7.907,Y -42.096,Z -81.654,A -90.000,B 90.000,C 0.000} C_DIS
LIN {X -7.717,Y -42.094,Z -81.636,A -90.000,B 90.000,C 0.000} C_DIS
LIN {X -7.498,Y -42.087,Z -81.617,A -90.000,B 90.000,C 0.000} C_DIS
LIN {X -6.845,Y -42.051,Z -81.565,A -90.000,B 90.000,C 0.000} C_DIS
LIN {X -5.709,Y -42.000,Z -81.512,A -90.000,B 90.000,C 0.000} C_DIS
LIN {X -5.489,Y -41.994,Z -81.509,A -90.000,B 90.000,C 0.000} C_DIS
LIN {X -4.530,Y -41.978,Z -81.537,A -90.000,B 90.000,C 0.000} C_DIS
LIN {X -4.239,Y -41.968,Z -81.544,A -90.000,B 90.000,C 0.000} C_DIS
LIN {X -2.478,Y -41.902,Z -81.592,A -90.000,B 90.000,C 0.000} C_DIS
LIN {X -2.330,Y -41.898,Z -81.600,A -90.000,B 90.000,C 0.000} C_DIS
LIN {X -1.928,Y -41.891,Z -81.630,A -90.000,B 90.000,C 0.000} C_DIS
LIN {X -1.610,Y -41.887,Z -81.659,A -90.000,B 90.000,C 0.000} C_DIS
LIN {X 0.111,Y -41.838,Z -81.826,A -90.000,B 90.000,C 0.000} C_DIS
LIN {X 0.666,Y -41.820,Z -81.880,A -90.000,B 90.000,C 0.000} C_DIS
LIN {X 1.033,Y -41.802,Z -81.914,A -90.000,B 90.000,C 0.000} C_DIS
LIN {X 1.251,Y -41.794,Z -81.942,A -90.000,B 90.000,C 0.000} C_DIS
LIN {X 2.014,Y -41.770,Z -82.047,A -90.000,B 90.000,C 0.000} C_DIS
LIN {X 4.449,Y -41.709,Z -82.439,A -90.000,B 90.000,C 0.000} C_DIS
LIN {X 4.855,Y -41.699,Z -82.511,A -90.000,B 90.000,C 0.000} C_DIS
LIN {X 5.215,Y -41.692,Z -82.581,A -90.000,B 90.000,C 0.000} C_DIS
LIN {X 6.675,Y -41.654,Z -82.840,A -90.000,B 90.000,C 0.000} C_DIS
LIN {X 7.311,Y -41.642,Z -82.951,A -90.000,B 90.000,C 0.000} C_DIS
LIN {X 7.804,Y -41.628,Z -83.040,A -90.000,B 90.000,C 0.000} C_DIS
LIN {X 8.920,Y -41.605,Z -83.264,A -90.000,B 90.000,C 0.000} C_DIS
LIN {X 10.132,Y -41.565,Z -83.485,A -90.000,B 90.000,C 0.000} C_DIS
LIN {X 10.383,Y -41.554,Z -83.532,A -90.000,B 90.000,C 0.000} C_DIS
LIN {X 10.546,Y -41.550,Z -83.562,A -90.000,B 90.000,C 0.000} C_DIS
LIN {X 12.198,Y -41.511,Z -83.876,A -90.000,B 90.000,C 0.000} C_DIS
LIN {X 12.848,Y -41.488,Z -83.987,A -90.000,B 90.000,C 0.000} C_DIS
LIN {X 13.407,Y -41.461,Z -84.087,A -90.000,B 90.000,C 0.000} C_DIS
LIN {X 14.740,Y -41.432,Z -84.300,A -90.000,B 90.000,C 0.000} C_DIS
LIN {X 15.283,Y -41.416,Z -84.389,A -90.000,B 90.000,C 0.000} C_DIS
LIN {X 15.654,Y -41.401,Z -84.444,A -90.000,B 90.000,C 0.000} C_DIS
LIN {X 16.259,Y -41.371,Z -84.524,A -90.000,B 90.000,C 0.000} C_DIS
LIN {X 16.822,Y -41.363,Z -84.590,A -90.000,B 90.000,C 0.000} C_DIS
LIN {X 17.208,Y -41.359,Z -84.634,A -90.000,B 90.000,C 0.000} C_DIS
LIN {X 18.224,Y -41.364,Z -84.771,A -90.000,B 90.000,C 0.000} C_DIS
LIN {X 18.369,Y -41.363,Z -84.788,A -90.000,B 90.000,C 0.000} C_DIS
LIN {X 19.145,Y -41.354,Z -84.867,A -90.000,B 90.000,C 0.000} C_DIS
LIN {X 20.423,Y -41.392,Z -84.965,A -90.000,B 90.000,C 0.000} C_DIS
LIN {X 20.820,Y -41.394,Z -84.980,A -90.000,B 90.000,C 0.000} C_DIS
LIN {X 21.005,Y -41.400,Z -84.983,A -90.000,B 90.000,C 0.000} C_DIS
LIN {X 21.291,Y -41.410,Z -84.990,A -90.000,B 90.000,C 0.000} C_DIS
LIN {X 21.991,Y -41.443,Z -85.018,A -90.000,B 90.000,C 0.000} C_DIS
LIN {X 22.907,Y -41.522,Z -85.037,A -90.000,B 90.000,C 0.000} C_DIS
LIN {X 23.931,Y -41.582,Z -84.992,A -90.000,B 90.000,C 0.000} C_DIS
LIN {X 24.365,Y -41.624,Z -84.965,A -90.000,B 90.000,C 0.000} C_DIS
LIN {X 24.676,Y -41.659,Z -84.944,A -90.000,B 90.000,C 0.000} C_DIS
LIN {X 24.861,Y -41.682,Z -84.938,A -90.000,B 90.000,C 0.000} C_DIS
LIN {X 25.145,Y -41.720,Z -84.939,A -90.000,B 90.000,C 0.000} C_DIS
LIN {X 25.482,Y -41.758,Z -84.913,A -90.000,B 90.000,C 0.000} C_DIS
LIN {X 27.067,Y -41.939,Z -84.809,A -90.000,B 90.000,C 0.000} C_DIS
LIN {X 27.755,Y -42.019,Z -84.766,A -90.000,B 90.000,C 0.000} C_DIS
LIN {X 27.861,Y -42.029,Z -84.759,A -90.000,B 90.000,C 0.000} C_DIS
LIN {X 28.204,Y -42.059,Z -84.711,A -90.000,B 90.000,C 0.000} C_DIS
LIN {X 28.344,Y -42.072,Z -84.695,A -90.000,B 90.000,C 0.000} C_DIS
LIN {X 28.548,Y -42.092,Z -84.682,A -90.000,B 90.000,C 0.000} C_DIS
LIN {X 28.983,Y -42.139,Z -84.670,A -90.000,B 90.000,C 0.000} C_DIS
LIN {X 29.309,Y -42.174,Z -84.663,A -90.000,B 90.000,C 0.000} C_DIS
LIN {X 31.094,Y -42.314,Z -84.643,A -90.000,B 90.000,C 0.000} C_DIS
LIN {X 31.364,Y -42.334,Z -84.640,A -90.000,B 90.000,C 0.000} C_DIS
LIN {X 32.037,Y -42.374,Z -84.570,A -90.000,B 90.000,C 0.000} C_DIS
LIN {X 32.228,Y -42.382,Z -84.551,A -90.000,B 90.000,C 0.000} C_DIS
LIN {X 32.370,Y -42.390,Z -84.542,A -90.000,B 90.000,C 0.000} C_DIS
LIN {X 32.595,Y -42.402,Z -84.534,A -90.000,B 90.000,C 0.000} C_DIS
LIN {X 32.888,Y -42.419,Z -84.531,A -90.000,B 90.000,C 0.000} C_DIS
LIN {X 32.961,Y -42.423,Z -84.533,A -90.000,B 90.000,C 0.000} C_DIS
LIN {X 33.270,Y -42.443,Z -84.545,A -90.000,B 90.000,C 0.000} C_DIS
LIN {X 33.422,Y -42.449,Z -84.552,A -90.000,B 90.000,C 0.000} C_DIS
LIN {X 34.271,Y -42.447,Z -84.598,A -90.000,B 90.000,C 0.000} C_DIS
LIN {X 34.487,Y -42.447,Z -84.616,A -90.000,B 90.000,C 0.000} C_DIS
LIN {X 34.624,Y -42.447,Z -84.633,A -90.000,B 90.000,C 0.000} C_DIS
LIN {X 34.863,Y -42.450,Z -84.675,A -90.000,B 90.000,C 0.000} C_DIS
LIN {X 35.206,Y -42.456,Z -84.744,A -90.000,B 90.000,C 0.000} C_DIS
LIN {X 36.133,Y -42.493,Z -84.927,A -90.000,B 90.000,C 0.000} C_DIS
LIN {X 36.220,Y -42.496,Z -84.945,A -90.000,B 90.000,C 0.000} C_DIS
LIN {X 36.803,Y -42.501,Z -85.064,A -90.000,B 90.000,C 0.000} C_DIS
LIN {X 37.061,Y -42.500,Z -85.100,A -90.000,B 90.000,C 0.000} C_DIS
LIN {X 37.243,Y -42.501,Z -85.133,A -90.000,B 90.000,C 0.000} C_DIS
LIN {X 37.542,Y -42.503,Z -85.195,A -90.000,B 90.000,C 0.000} C_DIS
LIN {X 37.851,Y -42.500,Z -85.275,A -90.000,B 90.000,C 0.000} C_DIS
LIN {X 38.159,Y -42.498,Z -85.369,A -90.000,B 90.000,C 0.000} C_DIS
LIN {X 38.442,Y -42.488,Z -85.461,A -90.000,B 90.000,C 0.000} C_DIS
LIN {X 39.673,Y -42.493,Z -85.847,A -90.000,B 90.000,C 0.000} C_DIS
LIN {X 39.752,Y -42.493,Z -85.872,A -90.000,B 90.000,C 0.000} C_DIS
LIN {X 40.014,Y -42.485,Z -85.958,A -90.000,B 90.000,C 0.000} C_DIS
LIN {X 40.193,Y -42.480,Z -86.026,A -90.000,B 90.000,C 0.000} C_DIS
LIN {X 40.292,Y -42.478,Z -86.067,A -90.000,B 90.000,C 0.000} C_DIS
LIN {X 40.565,Y -42.474,Z -86.187,A -90.000,B 90.000,C 0.000} C_DIS
LIN {X 41.042,Y -42.471,Z -86.414,A -90.000,B 90.000,C 0.000} C_DIS
LIN {X 41.531,Y -42.471,Z -86.645,A -90.000,B 90.000,C 0.000} C_DIS
LIN {X 41.930,Y -42.465,Z -86.835,A -90.000,B 90.000,C 0.000} C_DIS
LIN {X 42.291,Y -42.459,Z -87.010,A -90.000,B 90.000,C 0.000} C_DIS
LIN {X 42.532,Y -42.458,Z -87.143,A -90.000,B 90.000,C 0.000} C_DIS
LIN {X 42.851,Y -42.457,Z -87.323,A -90.000,B 90.000,C 0.000} C_DIS
LIN {X 42.971,Y -42.455,Z -87.396,A -90.000,B 90.000,C 0.000} C_DIS
LIN {X 43.153,Y -42.453,Z -87.519,A -90.000,B 90.000,C 0.000} C_DIS
LIN {X 43.458,Y -42.448,Z -87.742,A -90.000,B 90.000,C 0.000} C_DIS
LIN {X 44.195,Y -42.419,Z -88.162,A -90.000,B 90.000,C 0.000} C_DIS
LIN {X 44.541,Y -42.418,Z -88.356,A -90.000,B 90.000,C 0.000} C_DIS
LIN {X 44.684,Y -42.414,Z -88.438,A -90.000,B 90.000,C 0.000} C_DIS
LIN {X 44.902,Y -42.410,Z -88.578,A -90.000,B 90.000,C 0.000} C_DIS
LIN {X 45.046,Y -42.409,Z -88.679,A -90.000,B 90.000,C 0.000} C_DIS
LIN {X 45.308,Y -42.404,Z -88.870,A -90.000,B 90.000,C 0.000} C_DIS
LIN {X 46.179,Y -42.387,Z -89.516,A -90.000,B 90.000,C 0.000} C_DIS
LIN {X 46.361,Y -42.385,Z -89.663,A -90.000,B 90.000,C 0.000} C_DIS
LIN {X 47.120,Y -42.357,Z -90.304,A -90.000,B 90.000,C 0.000} C_DIS
LIN {X 47.190,Y -42.355,Z -90.365,A -90.000,B 90.000,C 0.000} C_DIS
LIN {X 47.306,Y -42.352,Z -90.472,A -90.000,B 90.000,C 0.000} C_DIS
LIN {X 47.404,Y -42.350,Z -90.570,A -90.000,B 90.000,C 0.000} C_DIS
LIN {X 47.476,Y -42.350,Z -90.647,A -90.000,B 90.000,C 0.000} C_DIS
LIN {X 48.065,Y -42.350,Z -91.295,A -90.000,B 90.000,C 0.000} C_DIS
LIN {X 48.358,Y -42.338,Z -91.624,A -90.000,B 90.000,C 0.000} C_DIS
LIN {X 48.865,Y -42.309,Z -92.124,A -90.000,B 90.000,C 0.000} C_DIS
LIN {X 48.999,Y -42.302,Z -92.265,A -90.000,B 90.000,C 0.000} C_DIS
LIN {X 49.198,Y -42.295,Z -92.489,A -90.000,B 90.000,C 0.000} C_DIS
LIN {X 49.313,Y -42.291,Z -92.626,A -90.000,B 90.000,C 0.000} C_DIS
LIN {X 49.703,Y -42.283,Z -93.120,A -90.000,B 90.000,C 0.000} C_DIS
LIN {X 49.788,Y -42.283,Z -93.236,A -90.000,B 90.000,C 0.000} C_DIS
LIN {X 49.949,Y -42.284,Z -93.471,A -90.000,B 90.000,C 0.000} C_DIS
LIN {X 50.041,Y -42.287,Z -93.620,A -90.000,B 90.000,C 0.000} C_DIS
LIN {X 50.425,Y -42.303,Z -94.281,A -90.000,B 90.000,C 0.000} C_DIS
LIN {X 50.543,Y -42.303,Z -94.488,A -90.000,B 90.000,C 0.000} C_DIS
LIN {X 51.262,Y -42.271,Z -95.764,A -90.000,B 90.000,C 0.000} C_DIS
LIN {X 51.891,Y -42.215,Z -96.897,A -90.000,B 90.000,C 0.000} C_DIS
LIN {X 51.941,Y -42.211,Z -96.993,A -90.000,B 90.000,C 0.000} C_DIS
LIN {X 52.066,Y -42.203,Z -97.252,A -90.000,B 90.000,C 0.000} C_DIS
LIN {X 52.424,Y -42.188,Z -98.097,A -90.000,B 90.000,C 0.000} C_DIS
LIN {X 52.506,Y -42.186,Z -98.314,A -90.000,B 90.000,C 0.000} C_DIS
LIN {X 52.734,Y -42.167,Z -99.010,A -90.000,B 90.000,C 0.000} C_DIS
LIN {X 52.792,Y -42.161,Z -99.216,A -90.000,B 90.000,C 0.000} C_DIS
LIN {X 52.884,Y -42.153,Z -99.571,A -90.000,B 90.000,C 0.000} C_DIS
LIN {X 53.033,Y -42.144,Z -100.199,A -90.000,B 90.000,C 0.000} C_DIS
LIN {X 53.100,Y -42.132,Z -100.496,A -90.000,B 90.000,C 0.000} C_DIS
LIN {X 53.461,Y -42.047,Z -102.109,A -90.000,B 90.000,C 0.000} C_DIS
LIN {X 53.487,Y -42.041,Z -102.248,A -90.000,B 90.000,C 0.000} C_DIS
LIN {X 53.530,Y -42.032,Z -102.526,A -90.000,B 90.000,C 0.000} C_DIS
LIN {X 53.546,Y -42.029,Z -102.665,A -90.000,B 90.000,C 0.000} C_DIS
LIN {X 53.712,Y -42.008,Z -104.614,A -90.000,B 90.000,C 0.000} C_DIS
LIN {X 53.722,Y -42.002,Z -104.752,A -90.000,B 90.000,C 0.000} C_DIS
LIN {X 53.792,Y -41.923,Z -105.859,A -90.000,B 90.000,C 0.000} C_DIS
LIN {X 53.827,Y -41.878,Z -106.447,A -90.000,B 90.000,C 0.000} C_DIS
LIN {X 53.831,Y -41.872,Z -106.538,A -90.000,B 90.000,C 0.000} C_DIS
LIN {X 53.834,Y -41.861,Z -106.722,A -90.000,B 90.000,C 0.000} C_DIS
LIN {X 53.833,Y -41.857,Z -106.817,A -90.000,B 90.000,C 0.000} C_DIS
LIN {X 53.817,Y -41.835,Z -107.392,A -90.000,B 90.000,C 0.000} C_DIS
LIN {X 53.804,Y -41.829,Z -107.610,A -90.000,B 90.000,C 0.000} C_DIS
LIN {X 53.785,Y -41.827,Z -107.807,A -90.000,B 90.000,C 0.000} C_DIS
LIN {X 53.721,Y -41.830,Z -108.295,A -90.000,B 90.000,C 0.000} C_DIS
LIN {X 53.665,Y -41.830,Z -108.787,A -90.000,B 90.000,C 0.000} C_DIS
LIN {X 53.302,Y -41.724,Z -111.587,A -90.000,B 90.000,C 0.000} C_DIS
LIN {X 53.284,Y -41.721,Z -111.706,A -90.000,B 90.000,C 0.000} C_DIS
LIN {X 53.221,Y -41.714,Z -112.069,A -90.000,B 90.000,C 0.000} C_DIS
LIN {X 53.171,Y -41.713,Z -112.312,A -90.000,B 90.000,C 0.000} C_DIS
LIN {X 53.078,Y -41.720,Z -112.711,A -90.000,B 90.000,C 0.000} C_DIS
LIN {X 53.008,Y -41.717,Z -112.999,A -90.000,B 90.000,C 0.000} C_DIS
LIN {X 52.857,Y -41.703,Z -113.597,A -90.000,B 90.000,C 0.000} C_DIS
LIN {X 52.449,Y -41.646,Z -115.187,A -90.000,B 90.000,C 0.000} C_DIS
LIN {X 52.328,Y -41.625,Z -115.680,A -90.000,B 90.000,C 0.000} C_DIS
LIN {X 52.251,Y -41.607,Z -115.982,A -90.000,B 90.000,C 0.000} C_DIS
LIN {X 52.213,Y -41.601,Z -116.117,A -90.000,B 90.000,C 0.000} C_DIS
LIN {X 52.153,Y -41.595,Z -116.312,A -90.000,B 90.000,C 0.000} C_DIS
LIN {X 52.116,Y -41.593,Z -116.420,A -90.000,B 90.000,C 0.000} C_DIS
LIN {X 51.954,Y -41.592,Z -116.862,A -90.000,B 90.000,C 0.000} C_DIS
LIN {X 51.872,Y -41.588,Z -117.080,A -90.000,B 90.000,C 0.000} C_DIS
LIN {X 51.702,Y -41.573,Z -117.524,A -90.000,B 90.000,C 0.000} C_DIS
LIN {X 51.094,Y -41.522,Z -119.103,A -90.000,B 90.000,C 0.000} C_DIS
LIN {X 50.663,Y -41.472,Z -120.190,A -90.000,B 90.000,C 0.000} C_DIS
LIN {X 50.598,Y -41.467,Z -120.343,A -90.000,B 90.000,C 0.000} C_DIS
LIN {X 50.457,Y -41.462,Z -120.651,A -90.000,B 90.000,C 0.000} C_DIS
LIN {X 50.364,Y -41.463,Z -120.839,A -90.000,B 90.000,C 0.000} C_DIS
LIN {X 50.204,Y -41.459,Z -121.129,A -90.000,B 90.000,C 0.000} C_DIS
LIN {X 50.051,Y -41.451,Z -121.402,A -90.000,B 90.000,C 0.000} C_DIS
LIN {X 49.731,Y -41.442,Z -121.952,A -90.000,B 90.000,C 0.000} C_DIS
LIN {X 48.355,Y -41.369,Z -124.268,A -90.000,B 90.000,C 0.000} C_DIS
LIN {X 48.211,Y -41.366,Z -124.495,A -90.000,B 90.000,C 0.000} C_DIS
LIN {X 48.142,Y -41.365,Z -124.603,A -90.000,B 90.000,C 0.000} C_DIS
LIN {X 48.004,Y -41.356,Z -124.801,A -90.000,B 90.000,C 0.000} C_DIS
LIN {X 47.937,Y -41.354,Z -124.891,A -90.000,B 90.000,C 0.000} C_DIS
LIN {X 47.642,Y -41.339,Z -125.248,A -90.000,B 90.000,C 0.000} C_DIS
LIN {X 47.046,Y -41.308,Z -125.965,A -90.000,B 90.000,C 0.000} C_DIS
LIN {X 47.046,Y -60.000,Z -125.965,A -90.000,B 90.000,C 0.000} C_DIS
LIN {X -74.102,Y -60.000,Z -243.561,A -90.000,B 90.000,C 0.000} C_DIS
LIN {X -74.102,Y -42.687,Z -243.561,A -90.000,B 90.000,C 0.000} C_DIS
LIN {X -74.090,Y -42.653,Z -243.496,A -90.000,B 90.000,C 0.000} C_DIS
LIN {X -74.027,Y -42.543,Z -243.275,A -90.000,B 90.000,C 0.000} C_DIS
LIN {X -73.956,Y -42.465,Z -243.102,A -90.000,B 90.000,C 0.000} C_DIS
LIN {X -73.924,Y -42.438,Z -243.037,A -90.000,B 90.000,C 0.000} C_DIS
LIN {X -73.882,Y -42.407,Z -242.959,A -90.000,B 90.000,C 0.000} C_DIS
LIN {X -73.856,Y -42.389,Z -242.914,A -90.000,B 90.000,C 0.000} C_DIS
LIN {X -73.650,Y -42.293,Z -242.630,A -90.000,B 90.000,C 0.000} C_DIS
LIN {X -73.511,Y -42.252,Z -242.480,A -90.000,B 90.000,C 0.000} C_DIS
LIN {X -73.414,Y -42.232,Z -242.390,A -90.000,B 90.000,C 0.000} C_DIS
LIN {X -73.306,Y -42.216,Z -242.302,A -90.000,B 90.000,C 0.000} C_DIS
LIN {X -73.011,Y -42.200,Z -242.107,A -90.000,B 90.000,C 0.000} C_DIS
LIN {X -70.995,Y -42.204,Z -240.982,A -90.000,B 90.000,C 0.000} C_DIS
LIN {X -69.430,Y -42.215,Z -240.120,A -90.000,B 90.000,C 0.000} C_DIS
LIN {X -68.671,Y -42.210,Z -239.711,A -90.000,B 90.000,C 0.000} C_DIS
LIN {X -68.083,Y -42.207,Z -239.396,A -90.000,B 90.000,C 0.000} C_DIS
LIN {X -66.074,Y -42.219,Z -238.360,A -90.000,B 90.000,C 0.000} C_DIS
LIN {X -62.859,Y -42.234,Z -236.696,A -90.000,B 90.000,C 0.000} C_DIS
LIN {X -60.671,Y -42.247,Z -235.562,A -90.000,B 90.000,C 0.000} C_DIS
LIN {X -59.684,Y -42.243,Z -235.058,A -90.000,B 90.000,C 0.000} C_DIS
LIN {X -57.194,Y -42.243,Z -233.825,A -90.000,B 90.000,C 0.000} C_DIS
LIN {X -54.435,Y -42.259,Z -232.489,A -90.000,B 90.000,C 0.000} C_DIS
LIN {X -52.618,Y -42.260,Z -231.618,A -90.000,B 90.000,C 0.000} C_DIS
LIN {X -51.585,Y -42.266,Z -231.133,A -90.000,B 90.000,C 0.000} C_DIS
LIN {X -48.900,Y -42.303,Z -229.911,A -90.000,B 90.000,C 0.000} C_DIS
LIN {X -46.187,Y -42.322,Z -228.688,A -90.000,B 90.000,C 0.000} C_DIS
LIN {X -43.905,Y -42.359,Z -227.698,A -90.000,B 90.000,C 0.000} C_DIS
LIN {X -42.479,Y -42.367,Z -227.089,A -90.000,B 90.000,C 0.000} C_DIS
LIN {X -40.513,Y -42.367,Z -226.229,A -90.000,B 90.000,C 0.000} C_DIS
LIN {X -38.028,Y -42.387,Z -225.183,A -90.000,B 90.000,C 0.000} C_DIS
LIN {X -37.446,Y -42.387,Z -224.941,A -90.000,B 90.000,C 0.000} C_DIS
LIN {X -37.134,Y -42.389,Z -224.814,A -90.000,B 90.000,C 0.000} C_DIS
LIN {X -35.442,Y -42.415,Z -224.165,A -90.000,B 90.000,C 0.000} C_DIS
LIN {X -35.302,Y -42.418,Z -224.110,A -90.000,B 90.000,C 0.000} C_DIS
LIN {X -33.811,Y -42.470,Z -223.562,A -90.000,B 90.000,C 0.000} C_DIS
LIN {X -33.408,Y -42.479,Z -223.405,A -90.000,B 90.000,C 0.000} C_DIS
LIN {X -30.871,Y -42.525,Z -222.419,A -90.000,B 90.000,C 0.000} C_DIS
LIN {X -30.569,Y -42.530,Z -222.307,A -90.000,B 90.000,C 0.000} C_DIS
LIN {X -28.736,Y -42.541,Z -221.638,A -90.000,B 90.000,C 0.000} C_DIS
LIN {X -27.656,Y -42.541,Z -221.246,A -90.000,B 90.000,C 0.000} C_DIS
LIN {X -26.403,Y -42.562,Z -220.782,A -90.000,B 90.000,C 0.000} C_DIS
LIN {X -26.050,Y -42.562,Z -220.636,A -90.000,B 90.000,C 0.000} C_DIS
LIN {X -25.938,Y -42.564,Z -220.596,A -90.000,B 90.000,C 0.000} C_DIS
LIN {X -24.877,Y -42.599,Z -220.249,A -90.000,B 90.000,C 0.000} C_DIS
LIN {X -20.995,Y -42.737,Z -219.001,A -90.000,B 90.000,C 0.000} C_DIS
LIN {X -20.611,Y -42.738,Z -218.882,A -90.000,B 90.000,C 0.000} C_DIS
LIN {X -19.457,Y -42.760,Z -218.519,A -90.000,B 90.000,C 0.000} C_DIS
LIN {X -18.618,Y -42.760,Z -218.205,A -90.000,B 90.000,C 0.000} C_DIS
LIN {X -17.439,Y -42.755,Z -217.743,A -90.000,B 90.000,C 0.000} C_DIS
LIN {X -17.158,Y -42.760,Z -217.656,A -90.000,B 90.000,C 0.000} C_DIS
LIN {X -17.008,Y -42.765,Z -217.620,A -90.000,B 90.000,C 0.000} C_DIS
LIN {X -15.119,Y -42.850,Z -217.193,A -90.000,B 90.000,C 0.000} C_DIS
LIN {X -14.356,Y -42.879,Z -217.002,A -90.000,B 90.000,C 0.000} C_DIS
LIN {X -14.013,Y -42.896,Z -216.914,A -90.000,B 90.000,C 0.000} C_DIS
LIN {X -13.471,Y -42.927,Z -216.776,A -90.000,B 90.000,C 0.000} C_DIS
LIN {X -12.882,Y -42.936,Z -216.631,A -90.000,B 90.000,C 0.000} C_DIS
LIN {X -12.370,Y -42.936,Z -216.469,A -90.000,B 90.000,C 0.000} C_DIS
LIN {X -11.750,Y -42.929,Z -216.237,A -90.000,B 90.000,C 0.000} C_DIS
LIN {X -10.902,Y -42.923,Z -215.935,A -90.000,B 90.000,C 0.000} C_DIS
LIN {X -10.619,Y -42.924,Z -215.834,A -90.000,B 90.000,C 0.000} C_DIS
LIN {X -10.539,Y -42.925,Z -215.807,A -90.000,B 90.000,C 0.000} C_DIS
LIN {X -10.422,Y -42.927,Z -215.774,A -90.000,B 90.000,C 0.000} C_DIS
LIN {X -10.224,Y -42.932,Z -215.725,A -90.000,B 90.000,C 0.000} C_DIS
LIN {X -9.958,Y -42.942,Z -215.681,A -90.000,B 90.000,C 0.000} C_DIS
LIN {X -8.696,Y -43.010,Z -215.572,A -90.000,B 90.000,C 0.000} C_DIS
LIN {X -8.277,Y -43.023,Z -215.488,A -90.000,B 90.000,C 0.000} C_DIS
LIN {X -7.362,Y -43.066,Z -215.302,A -90.000,B 90.000,C 0.000} C_DIS
LIN {X -6.828,Y -43.070,Z -215.197,A -90.000,B 90.000,C 0.000} C_DIS
LIN {X -6.536,Y -43.070,Z -215.122,A -90.000,B 90.000,C 0.000} C_DIS
LIN {X -5.933,Y -43.058,Z -214.868,A -90.000,B 90.000,C 0.000} C_DIS
LIN {X -5.686,Y -43.057,Z -214.791,A -90.000,B 90.000,C 0.000} C_DIS
LIN {X -5.511,Y -43.057,Z -214.748,A -90.000,B 90.000,C 0.000} C_DIS
LIN {X -5.370,Y -43.058,Z -214.719,A -90.000,B 90.000,C 0.000} C_DIS
LIN {X -5.173,Y -43.060,Z -214.686,A -90.000,B 90.000,C 0.000} C_DIS
LIN {X -4.720,Y -43.074,Z -214.608,A -90.000,B 90.000,C 0.000} C_DIS
LIN {X -4.593,Y -43.079,Z -214.591,A -90.000,B 90.000,C 0.000} C_DIS
LIN {X -4.286,Y -43.094,Z -214.582,A -90.000,B 90.000,C 0.000} C_DIS
LIN {X -3.262,Y -43.154,Z -214.631,A -90.000,B 90.000,C 0.000} C_DIS
LIN {X -3.005,Y -43.157,Z -214.548,A -90.000,B 90.000,C 0.000} C_DIS
LIN {X -2.453,Y -43.151,Z -214.370,A -90.000,B 90.000,C 0.000} C_DIS
LIN {X -1.501,Y -43.165,Z -214.062,A -90.000,B 90.000,C 0.000} C_DIS
LIN {X -0.854,Y -43.164,Z -213.704,A -90.000,B 90.000,C 0.000} C_DIS
LIN {X -0.651,Y -43.165,Z -213.610,A -90.000,B 90.000,C 0.000} C_DIS
LIN {X -0.593,Y -43.165,Z -213.586,A -90.000,B 90.000,C 0.000} C_DIS
LIN {X -0.237,Y -43.171,Z -213.477,A -90.000,B 90.000,C 0.000} C_DIS
LIN {X 1.172,Y -43.206,Z -213.196,A -90.000,B 90.000,C 0.000} C_DIS
LIN {X 2.063,Y -43.174,Z -212.299,A -90.000,B 90.000,C 0.000} C_DIS
LIN {X 2.419,Y -43.156,Z -211.941,A -90.000,B 90.000,C 0.000} C_DIS
LIN {X 2.556,Y -43.156,Z -211.803,A -90.000,B 90.000,C 0.000} C_DIS
LIN {X 2.620,Y -43.156,Z -211.741,A -90.000,B 90.000,C 0.000} C_DIS
LIN {X 3.391,Y -43.159,Z -211.028,A -90.000,B 90.000,C 0.000} C_DIS
LIN {X 4.865,Y -43.106,Z -208.847,A -90.000,B 90.000,C 0.000} C_DIS
LIN {X 5.327,Y -43.068,Z -208.169,A -90.000,B 90.000,C 0.000} C_DIS
LIN {X 5.389,Y -43.067,Z -208.080,A -90.000,B 90.000,C 0.000} C_DIS
LIN {X 6.592,Y -43.063,Z -206.430,A -90.000,B 90.000,C 0.000} C_DIS
LIN {X 6.982,Y -43.049,Z -205.735,A -90.000,B 90.000,C 0.000} C_DIS
LIN {X 7.872,Y -42.962,Z -204.168,A -90.000,B 90.000,C 0.000} C_DIS
LIN {X 8.474,Y -42.958,Z -203.154,A -90.000,B 90.000,C 0.000} C_DIS
LIN {X 9.111,Y -42.951,Z -202.079,A -90.000,B 90.000,C 0.000} C_DIS
LIN {X 9.868,Y -42.904,Z -200.820,A -90.000,B 90.000,C 0.000} C_DIS
LIN {X 10.128,Y -42.876,Z -200.305,A -90.000,B 90.000,C 0.000} C_DIS
LIN {X 10.252,Y -42.864,Z -200.070,A -90.000,B 90.000,C 0.000} C_DIS
LIN {X 11.134,Y -42.819,Z -198.382,A -90.000,B 90.000,C 0.000} C_DIS
LIN {X 11.277,Y -42.813,Z -198.125,A -90.000,B 90.000,C 0.000} C_DIS
LIN {X 11.847,Y -42.798,Z -197.146,A -90.000,B 90.000,C 0.000} C_DIS
LIN {X 12.581,Y -42.764,Z -195.892,A -90.000,B 90.000,C 0.000} C_DIS
LIN {X 12.735,Y -42.763,Z -195.647,A -90.000,B 90.000,C 0.000} C_DIS
LIN {X 12.804,Y -42.760,Z -195.522,A -90.000,B 90.000,C 0.000} C_DIS
LIN {X 13.272,Y -42.744,Z -194.703,A -90.000,B 90.000,C 0.000} C_DIS
LIN {X 14.825,Y -42.673,Z -192.005,A -90.000,B 90.000,C 0.000} C_DIS
LIN {X 14.930,Y -42.672,Z -191.842,A -90.000,B 90.000,C 0.000} C_DIS
LIN {X 15.790,Y -42.642,Z -190.553,A -90.000,B 90.000,C 0.000} C_DIS
LIN {X 17.121,Y -42.587,Z -188.354,A -90.000,B 90.000,C 0.000} C_DIS
LIN {X 17.272,Y -42.584,Z -188.119,A -90.000,B 90.000,C 0.000} C_DIS
LIN {X 17.371,Y -42.578,Z -187.975,A -90.000,B 90.000,C 0.000} C_DIS
LIN {X 18.423,Y -42.549,Z -186.547,A -90.000,B 90.000,C 0.000} C_DIS
LIN {X 18.568,Y -42.549,Z -186.348,A -90.000,B 90.000,C 0.000} C_DIS
LIN {X 19.594,Y -42.514,Z -184.821,A -90.000,B 90.000,C 0.000} C_DIS
LIN {X 19.623,Y -42.512,Z -184.779,A -90.000,B 90.000,C 0.000} C_DIS
LIN {X 19.712,Y -42.507,Z -184.658,A -90.000,B 90.000,C 0.000} C_DIS
LIN {X 20.843,Y -42.479,Z -183.236,A -90.000,B 90.000,C 0.000} C_DIS
LIN {X 21.182,Y -42.465,Z -182.814,A -90.000,B 90.000,C 0.000} C_DIS
LIN {X 21.975,Y -42.446,Z -181.889,A -90.000,B 90.000,C 0.000} C_DIS
LIN {X 23.280,Y -42.420,Z -180.417,A -90.000,B 90.000,C 0.000} C_DIS
LIN {X 24.142,Y -42.387,Z -179.456,A -90.000,B 90.000,C 0.000} C_DIS
LIN {X 24.311,Y -42.385,Z -179.274,A -90.000,B 90.000,C 0.000} C_DIS
LIN {X 25.050,Y -42.358,Z -178.440,A -90.000,B 90.000,C 0.000} C_DIS
LIN {X 25.914,Y -42.335,Z -177.484,A -90.000,B 90.000,C 0.000} C_DIS
LIN {X 26.172,Y -42.336,Z -177.192,A -90.000,B 90.000,C 0.000} C_DIS
LIN {X 26.357,Y -42.332,Z -176.971,A -90.000,B 90.000,C 0.000} C_DIS
LIN {X 27.619,Y -42.289,Z -175.482,A -90.000,B 90.000,C 0.000} C_DIS
LIN {X 27.824,Y -42.294,Z -175.233,A -90.000,B 90.000,C 0.000} C_DIS
LIN {X 28.461,Y -42.283,Z -174.391,A -90.000,B 90.000,C 0.000} C_DIS
LIN {X 29.048,Y -42.264,Z -173.624,A -90.000,B 90.000,C 0.000} C_DIS
LIN {X 29.138,Y -42.266,Z -173.502,A -90.000,B 90.000,C 0.000} C_DIS
LIN {X 29.420,Y -42.256,Z -173.079,A -90.000,B 90.000,C 0.000} C_DIS
LIN {X 29.993,Y -42.247,Z -172.245,A -90.000,B 90.000,C 0.000} C_DIS
LIN {X 30.363,Y -42.235,Z -171.714,A -90.000,B 90.000,C 0.000} C_DIS
LIN {X 30.521,Y -42.238,Z -171.478,A -90.000,B 90.000,C 0.000} C_DIS
LIN {X 31.091,Y -42.220,Z -170.554,A -90.000,B 90.000,C 0.000} C_DIS
LIN {X 31.564,Y -42.213,Z -169.809,A -90.000,B 90.000,C 0.000} C_DIS
LIN {X 31.712,Y -42.209,Z -169.579,A -90.000,B 90.000,C 0.000} C_DIS
LIN {X 31.859,Y -42.212,Z -169.341,A -90.000,B 90.000,C 0.000} C_DIS
LIN {X 32.142,Y -42.209,Z -168.850,A -90.000,B 90.000,C 0.000} C_DIS
LIN {X 32.682,Y -42.195,Z -167.924,A -90.000,B 90.000,C 0.000} C_DIS
LIN {X 32.992,Y -42.191,Z -167.403,A -90.000,B 90.000,C 0.000} C_DIS
LIN {X 33.187,Y -42.195,Z -167.068,A -90.000,B 90.000,C 0.000} C_DIS
LIN {X 33.789,Y -42.189,Z -165.988,A -90.000,B 90.000,C 0.000} C_DIS
LIN {X 34.416,Y -42.177,Z -164.874,A -90.000,B 90.000,C 0.000} C_DIS
LIN {X 34.528,Y -42.179,Z -164.673,A -90.000,B 90.000,C 0.000} C_DIS
LIN {X 35.172,Y -42.176,Z -163.476,A -90.000,B 90.000,C 0.000} C_DIS
LIN {X 35.642,Y -42.179,Z -162.617,A -90.000,B 90.000,C 0.000} C_DIS
LIN {X 35.886,Y -42.179,Z -162.175,A -90.000,B 90.000,C 0.000} C_DIS
LIN {X 36.046,Y -42.183,Z -161.876,A -90.000,B 90.000,C 0.000} C_DIS
LIN {X 36.392,Y -42.187,Z -161.216,A -90.000,B 90.000,C 0.000} C_DIS
LIN {X 37.384,Y -42.196,Z -159.349,A -90.000,B 90.000,C 0.000} C_DIS
LIN {X 37.616,Y -42.202,Z -158.907,A -90.000,B 90.000,C 0.000} C_DIS
LIN {X 38.795,Y -42.221,Z -156.618,A -90.000,B 90.000,C 0.000} C_DIS
LIN {X 39.178,Y -42.237,Z -155.859,A -90.000,B 90.000,C 0.000} C_DIS
LIN {X 39.477,Y -42.247,Z -155.263,A -90.000,B 90.000,C 0.000} C_DIS
LIN {X 40.033,Y -42.260,Z -154.179,A -90.000,B 90.000,C 0.000} C_DIS
LIN {X 40.132,Y -42.264,Z -153.990,A -90.000,B 90.000,C 0.000} C_DIS
LIN {X 40.489,Y -42.288,Z -153.295,A -90.000,B 90.000,C 0.000} C_DIS
LIN {X 40.715,Y -42.295,Z -152.865,A -90.000,B 90.000,C 0.000} C_DIS
LIN {X 41.267,Y -42.317,Z -151.833,A -90.000,B 90.000,C 0.000} C_DIS
LIN {X 41.553,Y -42.327,Z -151.306,A -90.000,B 90.000,C 0.000} C_DIS
LIN {X 41.711,Y -42.330,Z -151.022,A -90.000,B 90.000,C 0.000} C_DIS
LIN {X 42.047,Y -42.339,Z -150.413,A -90.000,B 90.000,C 0.000} C_DIS
LIN {X 42.357,Y -42.352,Z -149.866,A -90.000,B 90.000,C 0.000} C_DIS
LIN {X 42.627,Y -42.365,Z -149.399,A -90.000,B 90.000,C 0.000} C_DIS
LIN {X 42.707,Y -42.367,Z -149.262,A -90.000,B 90.000,C 0.000} C_DIS
LIN {X 43.291,Y -42.374,Z -148.273,A -90.000,B 90.000,C 0.000} C_DIS
LIN {X 44.042,Y -42.408,Z -147.055,A -90.000,B 90.000,C 0.000} C_DIS
LIN {X 44.460,Y -42.409,Z -146.394,A -90.000,B 90.000,C 0.000} C_DIS
LIN {X 44.779,Y -42.410,Z -145.901,A -90.000,B 90.000,C 0.000} C_DIS
LIN {X 44.821,Y -42.411,Z -145.838,A -90.000,B 90.000,C 0.000} C_DIS
LIN {X 45.309,Y -42.429,Z -145.136,A -90.000,B 90.000,C 0.000} C_DIS
LIN {X 45.541,Y -42.441,Z -144.822,A -90.000,B 90.000,C 0.000} C_DIS
LIN {X 46.934,Y -42.466,Z -142.979,A -90.000,B 90.000,C 0.000} C_DIS
LIN {X 46.988,Y -42.465,Z -142.910,A -90.000,B 90.000,C 0.000} C_DIS
LIN {X 47.079,Y -42.466,Z -142.800,A -90.000,B 90.000,C 0.000} C_DIS
LIN {X 47.814,Y -42.473,Z -141.918,A -90.000,B 90.000,C 0.000} C_DIS
LIN {X 48.043,Y -42.478,Z -141.651,A -90.000,B 90.000,C 0.000} C_DIS
LIN {X 48.510,Y -42.489,Z -141.127,A -90.000,B 90.000,C 0.000} C_DIS
LIN {X 48.862,Y -42.491,Z -140.736,A -90.000,B 90.000,C 0.000} C_DIS
LIN {X 48.962,Y -42.492,Z -140.629,A -90.000,B 90.000,C 0.000} C_DIS
LIN {X 49.930,Y -42.515,Z -139.629,A -90.000,B 90.000,C 0.000} C_DIS
LIN {X 50.330,Y -42.527,Z -139.225,A -90.000,B 90.000,C 0.000} C_DIS
LIN {X 51.369,Y -42.545,Z -138.208,A -90.000,B 90.000,C 0.000} C_DIS
LIN {X 51.617,Y -42.545,Z -137.968,A -90.000,B 90.000,C 0.000} C_DIS
LIN {X 52.449,Y -42.550,Z -137.180,A -90.000,B 90.000,C 0.000} C_DIS
LIN {X 52.832,Y -42.553,Z -136.817,A -90.000,B 90.000,C 0.000} C_DIS
LIN {X 52.917,Y -42.555,Z -136.741,A -90.000,B 90.000,C 0.000} C_DIS
LIN {X 53.403,Y -42.574,Z -136.327,A -90.000,B 90.000,C 0.000} C_DIS
LIN {X 53.954,Y -42.591,Z -135.841,A -90.000,B 90.000,C 0.000} C_DIS
LIN {X 55.073,Y -42.613,Z -134.831,A -90.000,B 90.000,C 0.000} C_DIS
LIN {X 55.463,Y -42.619,Z -134.472,A -90.000,B 90.000,C 0.000} C_DIS
LIN {X 56.119,Y -42.617,Z -133.873,A -90.000,B 90.000,C 0.000} C_DIS
LIN {X 56.267,Y -42.622,Z -133.736,A -90.000,B 90.000,C 0.000} C_DIS
LIN {X 56.378,Y -42.628,Z -133.640,A -90.000,B 90.000,C 0.000} C_DIS
LIN {X 56.784,Y -42.652,Z -133.306,A -90.000,B 90.000,C 0.000} C_DIS
LIN {X 57.100,Y -42.665,Z -133.022,A -90.000,B 90.000,C 0.000} C_DIS
LIN {X 58.239,Y -42.681,Z -131.869,A -90.000,B 90.000,C 0.000} C_DIS
LIN {X 58.712,Y -42.683,Z -131.372,A -90.000,B 90.000,C 0.000} C_DIS
LIN {X 59.142,Y -42.717,Z -130.905,A -90.000,B 90.000,C 0.000} C_DIS
LIN {X 59.830,Y -42.718,Z -129.864,A -90.000,B 90.000,C 0.000} C_DIS
LIN {X 60.555,Y -42.721,Z -128.767,A -90.000,B 90.000,C 0.000} C_DIS
LIN {X 61.400,Y -42.732,Z -127.509,A -90.000,B 90.000,C 0.000} C_DIS
LIN {X 61.425,Y -42.732,Z -127.472,A -90.000,B 90.000,C 0.000} C_DIS
LIN {X 61.586,Y -42.730,Z -127.210,A -90.000,B 90.000,C 0.000} C_DIS
LIN {X 62.079,Y -42.738,Z -126.401,A -90.000,B 90.000,C 0.000} C_DIS
LIN {X 62.158,Y -42.740,Z -126.282,A -90.000,B 90.000,C 0.000} C_DIS
LIN {X 62.201,Y -42.743,Z -126.224,A -90.000,B 90.000,C 0.000} C_DIS
LIN {X 62.266,Y -42.747,Z -126.142,A -90.000,B 90.000,C 0.000} C_DIS
LIN {X 62.388,Y -42.755,Z -125.999,A -90.000,B 90.000,C 0.000} C_DIS
LIN {X 62.486,Y -42.755,Z -125.891,A -90.000,B 90.000,C 0.000} C_DIS
LIN {X 62.549,Y -42.757,Z -125.827,A -90.000,B 90.000,C 0.000} C_DIS
LIN {X 63.001,Y -42.771,Z -125.403,A -90.000,B 90.000,C 0.000} C_DIS
LIN {X 63.044,Y -42.774,Z -125.361,A -90.000,B 90.000,C 0.000} C_DIS
LIN {X 64.214,Y -42.812,Z -123.940,A -90.000,B 90.000,C 0.000} C_DIS
LIN {X 64.464,Y -42.822,Z -123.646,A -90.000,B 90.000,C 0.000} C_DIS
LIN {X 64.556,Y -42.825,Z -123.546,A -90.000,B 90.000,C 0.000} C_DIS
LIN {X 64.700,Y -42.835,Z -123.413,A -90.000,B 90.000,C 0.000} C_DIS
LIN {X 64.770,Y -42.844,Z -123.356,A -90.000,B 90.000,C 0.000} C_DIS
LIN {X 64.959,Y -42.856,Z -123.209,A -90.000,B 90.000,C 0.000} C_DIS
LIN {X 65.128,Y -42.859,Z -123.097,A -90.000,B 90.000,C 0.000} C_DIS
LIN {X 65.197,Y -42.860,Z -123.059,A -90.000,B 90.000,C 0.000} C_DIS
LIN {X 67.556,Y -42.946,Z -121.882,A -90.000,B 90.000,C 0.000} C_DIS
LIN {X 67.752,Y -42.944,Z -121.734,A -90.000,B 90.000,C 0.000} C_DIS
LIN {X 67.843,Y -42.948,Z -121.664,A -90.000,B 90.000,C 0.000} C_DIS
LIN {X 67.949,Y -42.953,Z -121.587,A -90.000,B 90.000,C 0.000} C_DIS
LIN {X 68.006,Y -42.957,Z -121.550,A -90.000,B 90.000,C 0.000} C_DIS
LIN {X 68.219,Y -42.970,Z -121.425,A -90.000,B 90.000,C 0.000} C_DIS
LIN {X 68.354,Y -42.978,Z -121.353,A -90.000,B 90.000,C 0.000} C_DIS
LIN {X 68.397,Y -42.981,Z -121.333,A -90.000,B 90.000,C 0.000} C_DIS
LIN {X 68.514,Y -42.984,Z -121.286,A -90.000,B 90.000,C 0.000} C_DIS
LIN {X 68.561,Y -42.985,Z -121.269,A -90.000,B 90.000,C 0.000} C_DIS
LIN {X 68.683,Y -42.984,Z -121.232,A -90.000,B 90.000,C 0.000} C_DIS
LIN {X 68.732,Y -42.984,Z -121.220,A -90.000,B 90.000,C 0.000} C_DIS
LIN {X 68.898,Y -42.977,Z -121.181,A -90.000,B 90.000,C 0.000} C_DIS
LIN {X 69.043,Y -42.970,Z -121.152,A -90.000,B 90.000,C 0.000} C_DIS
LIN {X 69.085,Y -42.968,Z -121.146,A -90.000,B 90.000,C 0.000} C_DIS
LIN {X 69.458,Y -42.958,Z -121.129,A -90.000,B 90.000,C 0.000} C_DIS
LIN {X 69.625,Y -42.956,Z -121.136,A -90.000,B 90.000,C 0.000} C_DIS
LIN {X 69.894,Y -42.955,Z -121.158,A -90.000,B 90.000,C 0.000} C_DIS
LIN {X 70.106,Y -42.956,Z -121.189,A -90.000,B 90.000,C 0.000} C_DIS
LIN {X 70.207,Y -42.957,Z -121.210,A -90.000,B 90.000,C 0.000} C_DIS
LIN {X 71.040,Y -42.970,Z -121.384,A -90.000,B 90.000,C 0.000} C_DIS
LIN {X 71.130,Y -42.971,Z -121.404,A -90.000,B 90.000,C 0.000} C_DIS
LIN {X 71.992,Y -42.980,Z -121.609,A -90.000,B 90.000,C 0.000} C_DIS
LIN {X 72.151,Y -42.983,Z -121.653,A -90.000,B 90.000,C 0.000} C_DIS
LIN {X 72.394,Y -42.988,Z -121.734,A -90.000,B 90.000,C 0.000} C_DIS
LIN {X 73.018,Y -43.005,Z -121.964,A -90.000,B 90.000,C 0.000} C_DIS
LIN {X 73.190,Y -43.006,Z -122.028,A -90.000,B 90.000,C 0.000} C_DIS
LIN {X 73.763,Y -42.979,Z -122.247,A -90.000,B 90.000,C 0.000} C_DIS
LIN {X 74.408,Y -42.928,Z -122.498,A -90.000,B 90.000,C 0.000} C_DIS
LIN {X 74.801,Y -42.906,Z -122.708,A -90.000,B 90.000,C 0.000} C_DIS
LIN {X 74.875,Y -42.904,Z -122.759,A -90.000,B 90.000,C 0.000} C_DIS
LIN {X 75.030,Y -42.900,Z -122.869,A -90.000,B 90.000,C 0.000} C_DIS
LIN {X 75.218,Y -42.892,Z -123.007,A -90.000,B 90.000,C 0.000} C_DIS
LIN {X 75.496,Y -42.876,Z -123.214,A -90.000,B 90.000,C 0.000} C_DIS
LIN {X 75.594,Y -42.871,Z -123.295,A -90.000,B 90.000,C 0.000} C_DIS
LIN {X 75.636,Y -42.870,Z -123.332,A -90.000,B 90.000,C 0.000} C_DIS
LIN {X 75.827,Y -42.863,Z -123.526,A -90.000,B 90.000,C 0.000} C_DIS
LIN {X 76.032,Y -42.859,Z -123.751,A -90.000,B 90.000,C 0.000} C_DIS
LIN {X 76.203,Y -42.858,Z -123.968,A -90.000,B 90.000,C 0.000} C_DIS
LIN {X 76.264,Y -42.859,Z -124.058,A -90.000,B 90.000,C 0.000} C_DIS
LIN {X 76.711,Y -42.891,Z -124.705,A -90.000,B 90.000,C 0.000} C_DIS
LIN {X 76.841,Y -42.898,Z -124.894,A -90.000,B 90.000,C 0.000} C_DIS
LIN {X 77.170,Y -42.899,Z -125.381,A -90.000,B 90.000,C 0.000} C_DIS
LIN {X 77.291,Y -42.898,Z -125.584,A -90.000,B 90.000,C 0.000} C_DIS
LIN {X 77.367,Y -42.894,Z -125.722,A -90.000,B 90.000,C 0.000} C_DIS
LIN {X 77.407,Y -42.892,Z -125.803,A -90.000,B 90.000,C 0.000} C_DIS
LIN {X 77.465,Y -42.891,Z -125.940,A -90.000,B 90.000,C 0.000} C_DIS
LIN {X 77.632,Y -42.891,Z -126.381,A -90.000,B 90.000,C 0.000} C_DIS
LIN {X 77.766,Y -42.892,Z -126.755,A -90.000,B 90.000,C 0.000} C_DIS
LIN {X 77.983,Y -42.892,Z -127.362,A -90.000,B 90.000,C 0.000} C_DIS
LIN {X 78.054,Y -42.885,Z -127.567,A -90.000,B 90.000,C 0.000} C_DIS
LIN {X 78.143,Y -42.877,Z -127.842,A -90.000,B 90.000,C 0.000} C_DIS
LIN {X 78.195,Y -42.873,Z -128.036,A -90.000,B 90.000,C 0.000} C_DIS
LIN {X 78.342,Y -42.873,Z -128.821,A -90.000,B 90.000,C 0.000} C_DIS
LIN {X 78.359,Y -42.873,Z -128.917,A -90.000,B 90.000,C 0.000} C_DIS
LIN {X 78.420,Y -42.870,Z -129.328,A -90.000,B 90.000,C 0.000} C_DIS
LIN {X 78.512,Y -42.852,Z -129.970,A -90.000,B 90.000,C 0.000} C_DIS
LIN {X 78.522,Y -42.851,Z -130.054,A -90.000,B 90.000,C 0.000} C_DIS
LIN {X 78.546,Y -42.847,Z -130.290,A -90.000,B 90.000,C 0.000} C_DIS
LIN {X 78.638,Y -42.836,Z -131.414,A -90.000,B 90.000,C 0.000} C_DIS
LIN {X 78.735,Y -42.816,Z -132.396,A -90.000,B 90.000,C 0.000} C_DIS
LIN {X 78.824,Y -42.802,Z -133.825,A -90.000,B 90.000,C 0.000} C_DIS
LIN {X 78.876,Y -42.787,Z -134.347,A -90.000,B 90.000,C 0.000} C_DIS
LIN {X 79.021,Y -42.765,Z -135.771,A -90.000,B 90.000,C 0.000} C_DIS
LIN {X 79.099,Y -42.749,Z -136.329,A -90.000,B 90.000,C 0.000} C_DIS
LIN {X 79.159,Y -42.739,Z -136.890,A -90.000,B 90.000,C 0.000} C_DIS
LIN {X 79.270,Y -42.711,Z -137.979,A -90.000,B 90.000,C 0.000} C_DIS
LIN {X 79.426,Y -42.685,Z -139.477,A -90.000,B 90.000,C 0.000} C_DIS
LIN {X 79.459,Y -42.682,Z -139.919,A -90.000,B 90.000,C 0.000} C_DIS
LIN {X 79.474,Y -42.681,Z -140.155,A -90.000,B 90.000,C 0.000} C_DIS
LIN {X 79.592,Y -42.649,Z -142.220,A -90.000,B 90.000,C 0.000} C_DIS
LIN {X 79.638,Y -42.648,Z -143.459,A -90.000,B 90.000,C 0.000} C_DIS
LIN {X 79.639,Y -42.649,Z -143.553,A -90.000,B 90.000,C 0.000} C_DIS
LIN {X 79.637,Y -42.652,Z -143.806,A -90.000,B 90.000,C 0.000} C_DIS
LIN {X 79.648,Y -42.635,Z -146.504,A -90.000,B 90.000,C 0.000} C_DIS
LIN {X 79.652,Y -42.635,Z -147.209,A -90.000,B 90.000,C 0.000} C_DIS
LIN {X 79.650,Y -42.636,Z -147.307,A -90.000,B 90.000,C 0.000} C_DIS
LIN {X 79.645,Y -42.638,Z -147.444,A -90.000,B 90.000,C 0.000} C_DIS
LIN {X 79.602,Y -42.638,Z -148.379,A -90.000,B 90.000,C 0.000} C_DIS
LIN {X 79.493,Y -42.630,Z -151.273,A -90.000,B 90.000,C 0.000} C_DIS
LIN {X 79.483,Y -42.632,Z -151.400,A -90.000,B 90.000,C 0.000} C_DIS
LIN {X 79.359,Y -42.632,Z -152.794,A -90.000,B 90.000,C 0.000} C_DIS
LIN {X 79.156,Y -42.613,Z -155.135,A -90.000,B 90.000,C 0.000} C_DIS
LIN {X 79.144,Y -42.613,Z -155.240,A -90.000,B 90.000,C 0.000} C_DIS
LIN {X 79.127,Y -42.614,Z -155.361,A -90.000,B 90.000,C 0.000} C_DIS
LIN {X 78.906,Y -42.608,Z -156.922,A -90.000,B 90.000,C 0.000} C_DIS
LIN {X 78.832,Y -42.603,Z -157.439,A -90.000,B 90.000,C 0.000} C_DIS
LIN {X 78.607,Y -42.587,Z -159.015,A -90.000,B 90.000,C 0.000} C_DIS
LIN {X 78.578,Y -42.587,Z -159.190,A -90.000,B 90.000,C 0.000} C_DIS
LIN {X 78.549,Y -42.584,Z -159.352,A -90.000,B 90.000,C 0.000} C_DIS
LIN {X 77.824,Y -42.567,Z -162.846,A -90.000,B 90.000,C 0.000} C_DIS
LIN {X 77.775,Y -42.561,Z -163.074,A -90.000,B 90.000,C 0.000} C_DIS
LIN {X 77.756,Y -42.560,Z -163.156,A -90.000,B 90.000,C 0.000} C_DIS
LIN {X 76.749,Y -42.568,Z -166.643,A -90.000,B 90.000,C 0.000} C_DIS
LIN {X 76.706,Y -42.567,Z -166.782,A -90.000,B 90.000,C 0.000} C_DIS
LIN {X 75.586,Y -42.586,Z -170.085,A -90.000,B 90.000,C 0.000} C_DIS
LIN {X 74.915,Y -42.599,Z -171.992,A -90.000,B 90.000,C 0.000} C_DIS
LIN {X 74.646,Y -42.600,Z -172.753,A -90.000,B 90.000,C 0.000} C_DIS
LIN {X 74.472,Y -42.603,Z -173.245,A -90.000,B 90.000,C 0.000} C_DIS
LIN {X 73.581,Y -42.606,Z -176.015,A -90.000,B 90.000,C 0.000} C_DIS
LIN {X 73.537,Y -42.610,Z -176.158,A -90.000,B 90.000,C 0.000} C_DIS
LIN {X 72.944,Y -42.603,Z -178.630,A -90.000,B 90.000,C 0.000} C_DIS
LIN {X 72.879,Y -42.604,Z -178.907,A -90.000,B 90.000,C 0.000} C_DIS
LIN {X 72.447,Y -42.572,Z -181.311,A -90.000,B 90.000,C 0.000} C_DIS
LIN {X 72.376,Y -42.559,Z -181.804,A -90.000,B 90.000,C 0.000} C_DIS
LIN {X 72.080,Y -42.519,Z -183.900,A -90.000,B 90.000,C 0.000} C_DIS
LIN {X 71.951,Y -42.492,Z -184.877,A -90.000,B 90.000,C 0.000} C_DIS
LIN {X 71.749,Y -42.459,Z -186.440,A -90.000,B 90.000,C 0.000} C_DIS
LIN {X 71.710,Y -42.454,Z -186.722,A -90.000,B 90.000,C 0.000} C_DIS
LIN {X 71.668,Y -42.446,Z -187.006,A -90.000,B 90.000,C 0.000} C_DIS
LIN {X 71.534,Y -42.430,Z -187.828,A -90.000,B 90.000,C 0.000} C_DIS
LIN {X 71.311,Y -42.412,Z -189.212,A -90.000,B 90.000,C 0.000} C_DIS
LIN {X 71.137,Y -42.395,Z -190.104,A -90.000,B 90.000,C 0.000} C_DIS
LIN {X 71.007,Y -42.391,Z -190.693,A -90.000,B 90.000,C 0.000} C_DIS
LIN {X 70.765,Y -42.391,Z -191.801,A -90.000,B 90.000,C 0.000} C_DIS
LIN {X 70.746,Y -42.389,Z -191.888,A -90.000,B 90.000,C 0.000} C_DIS
LIN {X 70.220,Y -42.379,Z -193.880,A -90.000,B 90.000,C 0.000} C_DIS
LIN {X 69.940,Y -42.379,Z -194.952,A -90.000,B 90.000,C 0.000} C_DIS
LIN {X 69.889,Y -42.375,Z -195.134,A -90.000,B 90.000,C 0.000} C_DIS
LIN {X 69.718,Y -42.375,Z -195.679,A -90.000,B 90.000,C 0.000} C_DIS
LIN {X 69.191,Y -42.368,Z -197.398,A -90.000,B 90.000,C 0.000} C_DIS
LIN {X 68.937,Y -42.368,Z -198.232,A -90.000,B 90.000,C 0.000} C_DIS
LIN {X 68.874,Y -42.365,Z -198.431,A -90.000,B 90.000,C 0.000} C_DIS
LIN {X 68.545,Y -42.364,Z -199.374,A -90.000,B 90.000,C 0.000} C_DIS
LIN {X 67.851,Y -42.359,Z -201.386,A -90.000,B 90.000,C 0.000} C_DIS
LIN {X 67.598,Y -42.359,Z -202.119,A -90.000,B 90.000,C 0.000} C_DIS
LIN {X 67.516,Y -42.357,Z -202.353,A -90.000,B 90.000,C 0.000} C_DIS
LIN {X 67.122,Y -42.356,Z -203.407,A -90.000,B 90.000,C 0.000} C_DIS
LIN {X 66.045,Y -42.353,Z -206.300,A -90.000,B 90.000,C 0.000} C_DIS
LIN {X 65.901,Y -42.352,Z -206.685,A -90.000,B 90.000,C 0.000} C_DIS
LIN {X 64.108,Y -42.349,Z -211.249,A -90.000,B 90.000,C 0.000} C_DIS
LIN {X 63.908,Y -42.347,Z -211.753,A -90.000,B 90.000,C 0.000} C_DIS
LIN {X 63.326,Y -42.347,Z -213.166,A -90.000,B 90.000,C 0.000} C_DIS
LIN {X 62.141,Y -42.344,Z -216.056,A -90.000,B 90.000,C 0.000} C_DIS
LIN {X 61.814,Y -42.343,Z -216.852,A -90.000,B 90.000,C 0.000} C_DIS
LIN {X 60.421,Y -42.338,Z -220.124,A -90.000,B 90.000,C 0.000} C_DIS
LIN {X 59.706,Y -42.338,Z -221.792,A -90.000,B 90.000,C 0.000} C_DIS
LIN {X 59.594,Y -42.334,Z -222.049,A -90.000,B 90.000,C 0.000} C_DIS
LIN {X 57.275,Y -42.333,Z -227.069,A -90.000,B 90.000,C 0.000} C_DIS
LIN {X 57.122,Y -42.327,Z -227.389,A -90.000,B 90.000,C 0.000} C_DIS
LIN {X 55.577,Y -42.337,Z -230.370,A -90.000,B 90.000,C 0.000} C_DIS
LIN {X 54.555,Y -42.337,Z -232.367,A -90.000,B 90.000,C 0.000} C_DIS
LIN {X 54.352,Y -42.328,Z -232.750,A -90.000,B 90.000,C 0.000} C_DIS
LIN {X 54.176,Y -42.327,Z -233.055,A -90.000,B 90.000,C 0.000} C_DIS
LIN {X 52.440,Y -42.352,Z -235.953,A -90.000,B 90.000,C 0.000} C_DIS
LIN {X 51.296,Y -42.353,Z -237.922,A -90.000,B 90.000,C 0.000} C_DIS
LIN {X 51.070,Y -42.339,Z -238.296,A -90.000,B 90.000,C 0.000} C_DIS
LIN {X 50.975,Y -42.338,Z -238.441,A -90.000,B 90.000,C 0.000} C_DIS
LIN {X 48.956,Y -42.385,Z -241.279,A -90.000,B 90.000,C 0.000} C_DIS
LIN {X 47.772,Y -42.386,Z -243.033,A -90.000,B 90.000,C 0.000} C_DIS
LIN {X 47.477,Y -42.376,Z -243.459,A -90.000,B 90.000,C 0.000} C_DIS
LIN {X 47.402,Y -42.375,Z -243.561,A -90.000,B 90.000,C 0.000} C_DIS
LIN {X 47.402,Y -60.000,Z -243.561,A -90.000,B 90.000,C 0.000} C_DIS
LIN {X 40.115,Y -60.000,Z -150.353,A -90.000,B 90.000,C 0.000} C_DIS
LIN {X 40.115,Y -41.308,Z -150.353,A -90.000,B 90.000,C 0.000} C_DIS
LIN {X 40.550,Y -41.341,Z -149.540,A -90.000,B 90.000,C 0.000} C_DIS
LIN {X 40.704,Y -41.356,Z -149.259,A -90.000,B 90.000,C 0.000} C_DIS
LIN {X 40.866,Y -41.365,Z -148.971,A -90.000,B 90.000,C 0.000} C_DIS
LIN {X 41.075,Y -41.379,Z -148.603,A -90.000,B 90.000,C 0.000} C_DIS
LIN {X 41.791,Y -41.440,Z -147.337,A -90.000,B 90.000,C 0.000} C_DIS
LIN {X 41.882,Y -41.448,Z -147.184,A -90.000,B 90.000,C 0.000} C_DIS
LIN {X 42.658,Y -41.478,Z -145.931,A -90.000,B 90.000,C 0.000} C_DIS
LIN {X 43.060,Y -41.508,Z -145.272,A -90.000,B 90.000,C 0.000} C_DIS
LIN {X 43.323,Y -41.510,Z -144.867,A -90.000,B 90.000,C 0.000} C_DIS
LIN {X 43.664,Y -41.519,Z -144.377,A -90.000,B 90.000,C 0.000} C_DIS
LIN {X 43.860,Y -41.528,Z -144.093,A -90.000,B 90.000,C 0.000} C_DIS
LIN {X 44.557,Y -41.575,Z -143.141,A -90.000,B 90.000,C 0.000} C_DIS
LIN {X 45.600,Y -41.591,Z -141.766,A -90.000,B 90.000,C 0.000} C_DIS
LIN {X 45.950,Y -41.610,Z -141.333,A -90.000,B 90.000,C 0.000} C_DIS
LIN {X 46.048,Y -41.616,Z -141.211,A -90.000,B 90.000,C 0.000} C_DIS
LIN {X 46.279,Y -41.618,Z -140.935,A -90.000,B 90.000,C 0.000} C_DIS
LIN {X 46.499,Y -41.622,Z -140.672,A -90.000,B 90.000,C 0.000} C_DIS
LIN {X 46.700,Y -41.628,Z -140.438,A -90.000,B 90.000,C 0.000} C_DIS
LIN {X 47.541,Y -41.660,Z -139.484,A -90.000,B 90.000,C 0.000} C_DIS
LIN {X 47.673,Y -41.666,Z -139.342,A -90.000,B 90.000,C 0.000} C_DIS
LIN {X 48.646,Y -41.695,Z -138.334,A -90.000,B 90.000,C 0.000} C_DIS
LIN {X 49.060,Y -41.710,Z -137.914,A -90.000,B 90.000,C 0.000} C_DIS
LIN {X 49.675,Y -41.734,Z -137.303,A -90.000,B 90.000,C 0.000} C_DIS
LIN {X 49.982,Y -41.739,Z -137.003,A -90.000,B 90.000,C 0.000} C_DIS
LIN {X 50.410,Y -41.752,Z -136.582,A -90.000,B 90.000,C 0.000} C_DIS
LIN {X 51.460,Y -41.790,Z -135.570,A -90.000,B 90.000,C 0.000} C_DIS
LIN {X 51.624,Y -41.794,Z -135.416,A -90.000,B 90.000,C 0.000} C_DIS
LIN {X 51.733,Y -41.799,Z -135.317,A -90.000,B 90.000,C 0.000} C_DIS
LIN {X 52.204,Y -41.823,Z -134.913,A -90.000,B 90.000,C 0.000} C_DIS
LIN {X 52.730,Y -41.845,Z -134.447,A -90.000,B 90.000,C 0.000} C_DIS
LIN {X 53.531,Y -41.867,Z -133.720,A -90.000,B 90.000,C 0.000} C_DIS
LIN {X 53.703,Y -41.871,Z -133.564,A -90.000,B 90.000,C 0.000} C_DIS
LIN {X 53.965,Y -41.885,Z -133.320,A -90.000,B 90.000,C 0.000} C_DIS
LIN {X 55.000,Y -41.937,Z -132.348,A -90.000,B 90.000,C 0.000} C_DIS
LIN {X 55.164,Y -41.947,Z -132.203,A -90.000,B 90.000,C 0.000} C_DIS
LIN {X 55.575,Y -41.977,Z -131.861,A -90.000,B 90.000,C 0.000} C_DIS
LIN {X 55.810,Y -41.989,Z -131.649,A -90.000,B 90.000,C 0.000} C_DIS
LIN {X 56.770,Y -42.013,Z -130.673,A -90.000,B 90.000,C 0.000} C_DIS
LIN {X 56.886,Y -42.024,Z -130.551,A -90.000,B 90.000,C 0.000} C_DIS
LIN {X 57.517,Y -42.080,Z -129.862,A -90.000,B 90.000,C 0.000} C_DIS
LIN {X 57.651,Y -42.091,Z -129.716,A -90.000,B 90.000,C 0.000} C_DIS
LIN {X 58.595,Y -42.098,Z -128.285,A -90.000,B 90.000,C 0.000} C_DIS
LIN {X 58.978,Y -42.105,Z -127.702,A -90.000,B 90.000,C 0.000} C_DIS
LIN {X 59.826,Y -42.128,Z -126.433,A -90.000,B 90.000,C 0.000} C_DIS
LIN {X 60.108,Y -42.128,Z -125.972,A -90.000,B 90.000,C 0.000} C_DIS
LIN {X 60.492,Y -42.142,Z -125.341,A -90.000,B 90.000,C 0.000} C_DIS
LIN {X 60.569,Y -42.146,Z -125.223,A -90.000,B 90.000,C 0.000} C_DIS
LIN {X 60.672,Y -42.153,Z -125.076,A -90.000,B 90.000,C 0.000} C_DIS
LIN {X 60.791,Y -42.163,Z -124.924,A -90.000,B 90.000,C 0.000} C_DIS
LIN {X 60.874,Y -42.172,Z -124.825,A -90.000,B 90.000,C 0.000} C_DIS
LIN {X 61.062,Y -42.184,Z -124.607,A -90.000,B 90.000,C 0.000} C_DIS
LIN {X 61.165,Y -42.189,Z -124.499,A -90.000,B 90.000,C 0.000} C_DIS
LIN {X 61.247,Y -42.193,Z -124.418,A -90.000,B 90.000,C 0.000} C_DIS
LIN {X 61.648,Y -42.218,Z -124.036,A -90.000,B 90.000,C 0.000} C_DIS
LIN {X 61.770,Y -42.220,Z -123.888,A -90.000,B 90.000,C 0.000} C_DIS
LIN {X 62.764,Y -42.295,Z -122.663,A -90.000,B 90.000,C 0.000} C_DIS
LIN {X 63.048,Y -42.318,Z -122.327,A -90.000,B 90.000,C 0.000} C_DIS
LIN {X 63.141,Y -42.326,Z -122.223,A -90.000,B 90.000,C 0.000} C_DIS
LIN {X 63.257,Y -42.338,Z -122.105,A -90.000,B 90.000,C 0.000} C_DIS
LIN {X 63.465,Y -42.361,Z -121.912,A -90.000,B 90.000,C 0.000} C_DIS
LIN {X 63.690,Y -42.390,Z -121.731,A -90.000,B 90.000,C 0.000} C_DIS
LIN {X 63.817,Y -42.407,Z -121.631,A -90.000,B 90.000,C 0.000} C_DIS
LIN {X 63.890,Y -42.415,Z -121.578,A -90.000,B 90.000,C 0.000} C_DIS
LIN {X 64.070,Y -42.428,Z -121.456,A -90.000,B 90.000,C 0.000} C_DIS
LIN {X 64.207,Y -42.431,Z -121.374,A -90.000,B 90.000,C 0.000} C_DIS
LIN {X 64.337,Y -42.439,Z -121.303,A -90.000,B 90.000,C 0.000} C_DIS
LIN {X 64.478,Y -42.450,Z -121.231,A -90.000,B 90.000,C 0.000} C_DIS
LIN {X 66.516,Y -42.600,Z -120.198,A -90.000,B 90.000,C 0.000} C_DIS
LIN {X 66.710,Y -42.608,Z -120.051,A -90.000,B 90.000,C 0.000} C_DIS
LIN {X 66.806,Y -42.613,Z -119.982,A -90.000,B 90.000,C 0.000} C_DIS
LIN {X 66.945,Y -42.620,Z -119.888,A -90.000,B 90.000,C 0.000} C_DIS
LIN {X 67.114,Y -42.631,Z -119.786,A -90.000,B 90.000,C 0.000} C_DIS
LIN {X 67.287,Y -42.642,Z -119.686,A -90.000,B 90.000,C 0.000} C_DIS
LIN {X 67.445,Y -42.662,Z -119.600,A -90.000,B 90.000,C 0.000} C_DIS
LIN {X 67.591,Y -42.681,Z -119.528,A -90.000,B 90.000,C 0.000} C_DIS
LIN {X 67.715,Y -42.693,Z -119.474,A -90.000,B 90.000,C 0.000} C_DIS
LIN {X 67.855,Y -42.700,Z -119.419,A -90.000,B 90.000,C 0.000} C_DIS
LIN {X 68.004,Y -42.703,Z -119.369,A -90.000,B 90.000,C 0.000} C_DIS
LIN {X 68.197,Y -42.702,Z -119.313,A -90.000,B 90.000,C 0.000} C_DIS
LIN {X 68.432,Y -42.695,Z -119.256,A -90.000,B 90.000,C 0.000} C_DIS
LIN {X 68.647,Y -42.691,Z -119.212,A -90.000,B 90.000,C 0.000} C_DIS
LIN {X 68.783,Y -42.688,Z -119.188,A -90.000,B 90.000,C 0.000} C_DIS
LIN {X 68.891,Y -42.686,Z -119.175,A -90.000,B 90.000,C 0.000} C_DIS
LIN {X 68.991,Y -42.686,Z -119.168,A -90.000,B 90.000,C 0.000} C_DIS
LIN {X 69.363,Y -42.683,Z -119.150,A -90.000,B 90.000,C 0.000} C_DIS
LIN {X 69.469,Y -42.683,Z -119.148,A -90.000,B 90.000,C 0.000} C_DIS
LIN {X 69.705,Y -42.684,Z -119.156,A -90.000,B 90.000,C 0.000} C_DIS
LIN {X 69.963,Y -42.685,Z -119.176,A -90.000,B 90.000,C 0.000} C_DIS
LIN {X 70.116,Y -42.687,Z -119.189,A -90.000,B 90.000,C 0.000} C_DIS
LIN {X 70.393,Y -42.691,Z -119.228,A -90.000,B 90.000,C 0.000} C_DIS
LIN {X 70.550,Y -42.694,Z -119.256,A -90.000,B 90.000,C 0.000} C_DIS
LIN {X 71.532,Y -42.716,Z -119.461,A -90.000,B 90.000,C 0.000} C_DIS
LIN {X 71.823,Y -42.723,Z -119.530,A -90.000,B 90.000,C 0.000} C_DIS
LIN {X 72.499,Y -42.739,Z -119.689,A -90.000,B 90.000,C 0.000} C_DIS
LIN {X 72.629,Y -42.741,Z -119.725,A -90.000,B 90.000,C 0.000} C_DIS
LIN {X 72.734,Y -42.740,Z -119.756,A -90.000,B 90.000,C 0.000} C_DIS
LIN {X 72.870,Y -42.734,Z -119.802,A -90.000,B 90.000,C 0.000} C_DIS
LIN {X 73.104,Y -42.717,Z -119.884,A -90.000,B 90.000,C 0.000} C_DIS
LIN {X 75.139,Y -42.577,Z -120.670,A -90.000,B 90.000,C 0.000} C_DIS
LIN {X 75.176,Y -42.574,Z -120.685,A -90.000,B 90.000,C 0.000} C_DIS
LIN {X 75.323,Y -42.566,Z -120.756,A -90.000,B 90.000,C 0.000} C_DIS
LIN {X 75.764,Y -42.544,Z -120.993,A -90.000,B 90.000,C 0.000} C_DIS
LIN {X 75.859,Y -42.540,Z -121.051,A -90.000,B 90.000,C 0.000} C_DIS
LIN {X 76.030,Y -42.534,Z -121.169,A -90.000,B 90.000,C 0.000} C_DIS
LIN {X 76.272,Y -42.524,Z -121.343,A -90.000,B 90.000,C 0.000} C_DIS
LIN {X 76.669,Y -42.509,Z -121.635,A -90.000,B 90.000,C 0.000} C_DIS
LIN {X 76.838,Y -42.504,Z -121.773,A -90.000,B 90.000,C 0.000} C_DIS
LIN {X 76.950,Y -42.502,Z -121.870,A -90.000,B 90.000,C 0.000} C_DIS
LIN {X 77.028,Y -42.500,Z -121.945,A -90.000,B 90.000,C 0.000} C_DIS
LIN {X 77.226,Y -42.498,Z -122.145,A -90.000,B 90.000,C 0.000} C_DIS
LIN {X 77.481,Y -42.493,Z -122.422,A -90.000,B 90.000,C 0.000} C_DIS
LIN {X 77.576,Y -42.492,Z -122.534,A -90.000,B 90.000,C 0.000} C_DIS
LIN {X 77.773,Y -42.492,Z -122.785,A -90.000,B 90.000,C 0.000} C_DIS
LIN {X 77.886,Y -42.488,Z -122.949,A -90.000,B 90.000,C 0.000} C_DIS
LIN {X 77.973,Y -42.484,Z -123.077,A -90.000,B 90.000,C 0.000} C_DIS
LIN {X 78.108,Y -42.474,Z -123.280,A -90.000,B 90.000,C 0.000} C_DIS
LIN {X 78.799,Y -42.431,Z -124.319,A -90.000,B 90.000,C 0.000} C_DIS
LIN {X 78.921,Y -42.426,Z -124.523,A -90.000,B 90.000,C 0.000} C_DIS
LIN {X 78.964,Y -42.424,Z -124.597,A -90.000,B 90.000,C 0.000} C_DIS
LIN {X 79.061,Y -42.421,Z -124.769,A -90.000,B 90.000,C 0.000} C_DIS
LIN {X 79.147,Y -42.421,Z -124.937,A -90.000,B 90.000,C 0.000} C_DIS
LIN {X 79.181,Y -42.421,Z -125.008,A -90.000,B 90.000,C 0.000} C_DIS
LIN {X 79.274,Y -42.416,Z -125.233,A -90.000,B 90.000,C 0.000} C_DIS
LIN {X 79.486,Y -42.407,Z -125.802,A -90.000,B 90.000,C 0.000} C_DIS
LIN {X 79.693,Y -42.400,Z -126.387,A -90.000,B 90.000,C 0.000} C_DIS
LIN {X 79.889,Y -42.370,Z -126.958,A -90.000,B 90.000,C 0.000} C_DIS
LIN {X 79.981,Y -42.357,Z -127.247,A -90.000,B 90.000,C 0.000} C_DIS
LIN {X 80.038,Y -42.350,Z -127.457,A -90.000,B 90.000,C 0.000} C_DIS
LIN {X 80.080,Y -42.345,Z -127.627,A -90.000,B 90.000,C 0.000} C_DIS
LIN {X 80.180,Y -42.338,Z -128.167,A -90.000,B 90.000,C 0.000} C_DIS
LIN {X 80.202,Y -42.335,Z -128.286,A -90.000,B 90.000,C 0.000} C_DIS
LIN {X 80.260,Y -42.322,Z -128.631,A -90.000,B 90.000,C 0.000} C_DIS
LIN {X 80.415,Y -42.291,Z -129.720,A -90.000,B 90.000,C 0.000} C_DIS
LIN {X 80.459,Y -42.284,Z -130.134,A -90.000,B 90.000,C 0.000} C_DIS
LIN {X 80.491,Y -42.276,Z -130.540,A -90.000,B 90.000,C 0.000} C_DIS
LIN {X 80.544,Y -42.258,Z -131.234,A -90.000,B 90.000,C 0.000} C_DIS
LIN {X 80.571,Y -42.249,Z -131.511,A -90.000,B 90.000,C 0.000} C_DIS
LIN {X 80.640,Y -42.235,Z -132.218,A -90.000,B 90.000,C 0.000} C_DIS
LIN {X 80.658,Y -42.232,Z -132.495,A -90.000,B 90.000,C 0.000} C_DIS
LIN {X 80.727,Y -42.206,Z -133.671,A -90.000,B 90.000,C 0.000} C_DIS
LIN {X 80.777,Y -42.190,Z -134.177,A -90.000,B 90.000,C 0.000} C_DIS
LIN {X 80.913,Y -42.154,Z -135.552,A -90.000,B 90.000,C 0.000} C_DIS
LIN {X 80.990,Y -42.133,Z -136.116,A -90.000,B 90.000,C 0.000} C_DIS
LIN {X 81.017,Y -42.126,Z -136.380,A -90.000,B 90.000,C 0.000} C_DIS
LIN {X 81.091,Y -42.112,Z -137.086,A -90.000,B 90.000,C 0.000} C_DIS
LIN {X 81.135,Y -42.101,Z -137.512,A -90.000,B 90.000,C 0.000} C_DIS
LIN {X 81.318,Y -42.054,Z -139.329,A -90.000,B 90.000,C 0.000} C_DIS
LIN {X 81.356,Y -42.045,Z -139.868,A -90.000,B 90.000,C 0.000} C_DIS
LIN {X 81.477,Y -41.983,Z -142.150,A -90.000,B 90.000,C 0.000} C_DIS
LIN {X 81.502,Y -41.966,Z -142.994,A -90.000,B 90.000,C 0.000} C_DIS
LIN {X 81.514,Y -41.956,Z -143.438,A -90.000,B 90.000,C 0.000} C_DIS
LIN {X 81.515,Y -41.955,Z -143.579,A -90.000,B 90.000,C 0.000} C_DIS
LIN {X 81.511,Y -41.953,Z -143.888,A -90.000,B 90.000,C 0.000} C_DIS
LIN {X 81.510,Y -41.943,Z -144.324,A -90.000,B 90.000,C 0.000} C_DIS
LIN {X 81.505,Y -41.883,Z -147.247,A -90.000,B 90.000,C 0.000} C_DIS
LIN {X 81.500,Y -41.882,Z -147.408,A -90.000,B 90.000,C 0.000} C_DIS
LIN {X 81.489,Y -41.882,Z -147.654,A -90.000,B 90.000,C 0.000} C_DIS
LIN {X 81.446,Y -41.868,Z -148.455,A -90.000,B 90.000,C 0.000} C_DIS
LIN {X 81.318,Y -41.819,Z -151.376,A -90.000,B 90.000,C 0.000} C_DIS
LIN {X 81.281,Y -41.817,Z -151.801,A -90.000,B 90.000,C 0.000} C_DIS
LIN {X 81.171,Y -41.800,Z -152.950,A -90.000,B 90.000,C 0.000} C_DIS
LIN {X 80.962,Y -41.767,Z -155.285,A -90.000,B 90.000,C 0.000} C_DIS
LIN {X 80.938,Y -41.766,Z -155.494,A -90.000,B 90.000,C 0.000} C_DIS
LIN {X 80.917,Y -41.767,Z -155.643,A -90.000,B 90.000,C 0.000} C_DIS
LIN {X 80.540,Y -41.739,Z -158.256,A -90.000,B 90.000,C 0.000} C_DIS
LIN {X 80.389,Y -41.728,Z -159.311,A -90.000,B 90.000,C 0.000} C_DIS
LIN {X 80.358,Y -41.726,Z -159.491,A -90.000,B 90.000,C 0.000} C_DIS
LIN {X 80.317,Y -41.722,Z -159.714,A -90.000,B 90.000,C 0.000} C_DIS
LIN {X 79.889,Y -41.710,Z -161.774,A -90.000,B 90.000,C 0.000} C_DIS
LIN {X 79.628,Y -41.704,Z -163.034,A -90.000,B 90.000,C 0.000} C_DIS
LIN {X 79.522,Y -41.692,Z -163.516,A -90.000,B 90.000,C 0.000} C_DIS
LIN {X 79.486,Y -41.690,Z -163.658,A -90.000,B 90.000,C 0.000} C_DIS
LIN {X 78.566,Y -41.697,Z -166.839,A -90.000,B 90.000,C 0.000} C_DIS
LIN {X 78.426,Y -41.692,Z -167.306,A -90.000,B 90.000,C 0.000} C_DIS
LIN {X 77.406,Y -41.711,Z -170.318,A -90.000,B 90.000,C 0.000} C_DIS
LIN {X 77.280,Y -41.711,Z -170.686,A -90.000,B 90.000,C 0.000} C_DIS
LIN {X 76.341,Y -41.729,Z -173.360,A -90.000,B 90.000,C 0.000} C_DIS
LIN {X 76.180,Y -41.736,Z -173.823,A -90.000,B 90.000,C 0.000} C_DIS
LIN {X 75.363,Y -41.742,Z -176.365,A -90.000,B 90.000,C 0.000} C_DIS
LIN {X 75.276,Y -41.748,Z -176.647,A -90.000,B 90.000,C 0.000} C_DIS
LIN {X 74.906,Y -41.736,Z -178.173,A -90.000,B 90.000,C 0.000} C_DIS
LIN {X 74.696,Y -41.732,Z -179.047,A -90.000,B 90.000,C 0.000} C_DIS
LIN {X 74.643,Y -41.733,Z -179.271,A -90.000,B 90.000,C 0.000} C_DIS
LIN {X 74.342,Y -41.705,Z -180.931,A -90.000,B 90.000,C 0.000} C_DIS
LIN {X 74.225,Y -41.696,Z -181.582,A -90.000,B 90.000,C 0.000} C_DIS
LIN {X 73.910,Y -41.641,Z -183.767,A -90.000,B 90.000,C 0.000} C_DIS
LIN {X 73.860,Y -41.635,Z -184.122,A -90.000,B 90.000,C 0.000} C_DIS
LIN {X 73.754,Y -41.613,Z -184.930,A -90.000,B 90.000,C 0.000} C_DIS
LIN {X 73.516,Y -41.564,Z -186.720,A -90.000,B 90.000,C 0.000} C_DIS
LIN {X 73.459,Y -41.555,Z -187.124,A -90.000,B 90.000,C 0.000} C_DIS
LIN {X 73.409,Y -41.548,Z -187.445,A -90.000,B 90.000,C 0.000} C_DIS
LIN {X 73.246,Y -41.528,Z -188.434,A -90.000,B 90.000,C 0.000} C_DIS
LIN {X 73.059,Y -41.500,Z -189.548,A -90.000,B 90.000,C 0.000} C_DIS
LIN {X 72.874,Y -41.479,Z -190.481,A -90.000,B 90.000,C 0.000} C_DIS
LIN {X 72.604,Y -41.466,Z -191.695,A -90.000,B 90.000,C 0.000} C_DIS
LIN {X 72.456,Y -41.453,Z -192.334,A -90.000,B 90.000,C 0.000} C_DIS
LIN {X 71.622,Y -41.403,Z -195.418,A -90.000,B 90.000,C 0.000} C_DIS
LIN {X 71.553,Y -41.396,Z -195.656,A -90.000,B 90.000,C 0.000} C_DIS
LIN {X 71.339,Y -41.391,Z -196.333,A -90.000,B 90.000,C 0.000} C_DIS
LIN {X 71.116,Y -41.380,Z -197.045,A -90.000,B 90.000,C 0.000} C_DIS
LIN {X 70.584,Y -41.352,Z -198.734,A -90.000,B 90.000,C 0.000} C_DIS
LIN {X 70.498,Y -41.344,Z -198.997,A -90.000,B 90.000,C 0.000} C_DIS
LIN {X 70.002,Y -41.331,Z -200.403,A -90.000,B 90.000,C 0.000} C_DIS
LIN {X 69.272,Y -41.308,Z -202.485,A -90.000,B 90.000,C 0.000} C_DIS
LIN {X 69.272,Y -60.000,Z -202.485,A -90.000,B 90.000,C 0.000} C_DIS
LIN {X -45.739,Y -60.000,Z -226.626,A -90.000,B 90.000,C 0.000} C_DIS
LIN {X -45.739,Y -41.308,Z -226.626,A -90.000,B 90.000,C 0.000} C_DIS
LIN {X -44.574,Y -41.330,Z -226.119,A -90.000,B 90.000,C 0.000} C_DIS
LIN {X -43.161,Y -41.357,Z -225.503,A -90.000,B 90.000,C 0.000} C_DIS
LIN {X -41.732,Y -41.378,Z -224.865,A -90.000,B 90.000,C 0.000} C_DIS
LIN {X -41.182,Y -41.382,Z -224.622,A -90.000,B 90.000,C 0.000} C_DIS
LIN {X -38.047,Y -41.436,Z -223.286,A -90.000,B 90.000,C 0.000} C_DIS
LIN {X -37.753,Y -41.443,Z -223.164,A -90.000,B 90.000,C 0.000} C_DIS
LIN {X -36.819,Y -41.476,Z -222.795,A -90.000,B 90.000,C 0.000} C_DIS
LIN {X -36.066,Y -41.500,Z -222.499,A -90.000,B 90.000,C 0.000} C_DIS
LIN {X -35.888,Y -41.506,Z -222.430,A -90.000,B 90.000,C 0.000} C_DIS
LIN {X -35.068,Y -41.539,Z -222.126,A -90.000,B 90.000,C 0.000} C_DIS
LIN {X -34.420,Y -41.561,Z -221.888,A -90.000,B 90.000,C 0.000} C_DIS
LIN {X -31.681,Y -41.624,Z -220.816,A -90.000,B 90.000,C 0.000} C_DIS
LIN {X -31.480,Y -41.628,Z -220.738,A -90.000,B 90.000,C 0.000} C_DIS
LIN {X -29.476,Y -41.677,Z -219.987,A -90.000,B 90.000,C 0.000} C_DIS
LIN {X -27.048,Y -41.772,Z -219.061,A -90.000,B 90.000,C 0.000} C_DIS
LIN {X -26.754,Y -41.778,Z -218.936,A -90.000,B 90.000,C 0.000} C_DIS
LIN {X -26.656,Y -41.781,Z -218.897,A -90.000,B 90.000,C 0.000} C_DIS
LIN {X -26.488,Y -41.789,Z -218.836,A -90.000,B 90.000,C 0.000} C_DIS
LIN {X -25.526,Y -41.846,Z -218.510,A -90.000,B 90.000,C 0.000} C_DIS
LIN {X -24.146,Y -41.900,Z -218.064,A -90.000,B 90.000,C 0.000} C_DIS
LIN {X -22.564,Y -41.956,Z -217.556,A -90.000,B 90.000,C 0.000} C_DIS
LIN {X -20.135,Y -42.078,Z -216.760,A -90.000,B 90.000,C 0.000} C_DIS
LIN {X -20.063,Y -42.081,Z -216.737,A -90.000,B 90.000,C 0.000} C_DIS
LIN {X -19.217,Y -42.110,Z -216.408,A -90.000,B 90.000,C 0.000} C_DIS
LIN {X -18.135,Y -42.142,Z -215.971,A -90.000,B 90.000,C 0.000} C_DIS
LIN {X -17.996,Y -42.148,Z -215.921,A -90.000,B 90.000,C 0.000} C_DIS
LIN {X -17.718,Y -42.164,Z -215.830,A -90.000,B 90.000,C 0.000} C_DIS
LIN {X -17.576,Y -42.174,Z -215.790,A -90.000,B 90.000,C 0.000} C_DIS
LIN {X -17.406,Y -42.188,Z -215.747,A -90.000,B 90.000,C 0.000} C_DIS
LIN {X -16.817,Y -42.240,Z -215.606,A -90.000,B 90.000,C 0.000} C_DIS
LIN {X -16.291,Y -42.264,Z -215.487,A -90.000,B 90.000,C 0.000} C_DIS
LIN {X -15.826,Y -42.294,Z -215.379,A -90.000,B 90.000,C 0.000} C_DIS
LIN {X -15.544,Y -42.310,Z -215.314,A -90.000,B 90.000,C 0.000} C_DIS
LIN {X -13.395,Y -42.419,Z -214.768,A -90.000,B 90.000,C 0.000} C_DIS
LIN {X -13.003,Y -42.434,Z -214.638,A -90.000,B 90.000,C 0.000} C_DIS
LIN {X -12.346,Y -42.452,Z -214.387,A -90.000,B 90.000,C 0.000} C_DIS
LIN {X -11.236,Y -42.488,Z -213.982,A -90.000,B 90.000,C 0.000} C_DIS
LIN {X -11.156,Y -42.491,Z -213.955,A -90.000,B 90.000,C 0.000} C_DIS
LIN {X -10.941,Y -42.501,Z -213.890,A -90.000,B 90.000,C 0.000} C_DIS
LIN {X -10.663,Y -42.518,Z -213.818,A -90.000,B 90.000,C 0.000} C_DIS
LIN {X -10.529,Y -42.529,Z -213.790,A -90.000,B 90.000,C 0.000} C_DIS
LIN {X -10.264,Y -42.553,Z -213.743,A -90.000,B 90.000,C 0.000} C_DIS
LIN {X -10.107,Y -42.570,Z -213.722,A -90.000,B 90.000,C 0.000} C_DIS
LIN {X -8.959,Y -42.640,Z -213.621,A -90.000,B 90.000,C 0.000} C_DIS
LIN {X -7.574,Y -42.696,Z -213.341,A -90.000,B 90.000,C 0.000} C_DIS
LIN {X -7.262,Y -42.713,Z -213.277,A -90.000,B 90.000,C 0.000} C_DIS
LIN {X -7.170,Y -42.717,Z -213.252,A -90.000,B 90.000,C 0.000} C_DIS
LIN {X -6.641,Y -42.725,Z -213.027,A -90.000,B 90.000,C 0.000} C_DIS
LIN {X -6.524,Y -42.729,Z -212.986,A -90.000,B 90.000,C 0.000} C_DIS
LIN {X -6.277,Y -42.737,Z -212.907,A -90.000,B 90.000,C 0.000} C_DIS
LIN {X -6.192,Y -42.741,Z -212.882,A -90.000,B 90.000,C 0.000} C_DIS
LIN {X -5.903,Y -42.755,Z -212.810,A -90.000,B 90.000,C 0.000} C_DIS
LIN {X -5.697,Y -42.766,Z -212.768,A -90.000,B 90.000,C 0.000} C_DIS
LIN {X -5.270,Y -42.791,Z -212.693,A -90.000,B 90.000,C 0.000} C_DIS
LIN {X -4.983,Y -42.807,Z -212.644,A -90.000,B 90.000,C 0.000} C_DIS
LIN {X -4.807,Y -42.817,Z -212.619,A -90.000,B 90.000,C 0.000} C_DIS
LIN {X -4.638,Y -42.829,Z -212.607,A -90.000,B 90.000,C 0.000} C_DIS
LIN {X -4.383,Y -42.845,Z -212.599,A -90.000,B 90.000,C 0.000} C_DIS
LIN {X -4.332,Y -42.848,Z -212.597,A -90.000,B 90.000,C 0.000} C_DIS
LIN {X -4.166,Y -42.859,Z -212.599,A -90.000,B 90.000,C 0.000} C_DIS
LIN {X -3.520,Y -42.902,Z -212.630,A -90.000,B 90.000,C 0.000} C_DIS
LIN {X -2.294,Y -42.932,Z -212.231,A -90.000,B 90.000,C 0.000} C_DIS
LIN {X -1.816,Y -42.932,Z -211.966,A -90.000,B 90.000,C 0.000} C_DIS
LIN {X -1.688,Y -42.932,Z -211.901,A -90.000,B 90.000,C 0.000} C_DIS
LIN {X -1.428,Y -42.935,Z -211.781,A -90.000,B 90.000,C 0.000} C_DIS
LIN {X -1.352,Y -42.936,Z -211.750,A -90.000,B 90.000,C 0.000} C_DIS
LIN {X -1.172,Y -42.940,Z -211.685,A -90.000,B 90.000,C 0.000} C_DIS
LIN {X -0.817,Y -42.949,Z -211.576,A -90.000,B 90.000,C 0.000} C_DIS
LIN {X -0.621,Y -42.956,Z -211.526,A -90.000,B 90.000,C 0.000} C_DIS
LIN {X 0.188,Y -42.986,Z -211.364,A -90.000,B 90.000,C 0.000} C_DIS
LIN {X 0.766,Y -42.956,Z -210.783,A -90.000,B 90.000,C 0.000} C_DIS
LIN {X 1.029,Y -42.954,Z -210.517,A -90.000,B 90.000,C 0.000} C_DIS
LIN {X 1.215,Y -42.949,Z -210.332,A -90.000,B 90.000,C 0.000} C_DIS
LIN {X 1.871,Y -42.937,Z -209.726,A -90.000,B 90.000,C 0.000} C_DIS
LIN {X 3.526,Y -42.800,Z -207.296,A -90.000,B 90.000,C 0.000} C_DIS
LIN {X 3.706,Y -42.779,Z -207.033,A -90.000,B 90.000,C 0.000} C_DIS
LIN {X 3.790,Y -42.774,Z -206.914,A -90.000,B 90.000,C 0.000} C_DIS
LIN {X 4.929,Y -42.724,Z -205.366,A -90.000,B 90.000,C 0.000} C_DIS
LIN {X 5.575,Y -42.662,Z -204.228,A -90.000,B 90.000,C 0.000} C_DIS
LIN {X 5.942,Y -42.624,Z -203.583,A -90.000,B 90.000,C 0.000} C_DIS
LIN {X 6.182,Y -42.588,Z -203.167,A -90.000,B 90.000,C 0.000} C_DIS
LIN {X 6.256,Y -42.579,Z -203.045,A -90.000,B 90.000,C 0.000} C_DIS
LIN {X 7.681,Y -42.496,Z -200.672,A -90.000,B 90.000,C 0.000} C_DIS
LIN {X 8.159,Y -42.445,Z -199.884,A -90.000,B 90.000,C 0.000} C_DIS
LIN {X 8.399,Y -42.406,Z -199.418,A -90.000,B 90.000,C 0.000} C_DIS
LIN {X 8.597,Y -42.377,Z -199.048,A -90.000,B 90.000,C 0.000} C_DIS
LIN {X 9.444,Y -42.290,Z -197.453,A -90.000,B 90.000,C 0.000} C_DIS
LIN {X 9.608,Y -42.277,Z -197.162,A -90.000,B 90.000,C 0.000} C_DIS
LIN {X 10.821,Y -42.190,Z -195.109,A -90.000,B 90.000,C 0.000} C_DIS
LIN {X 10.931,Y -42.185,Z -194.922,A -90.000,B 90.000,C 0.000} C_DIS
LIN {X 11.081,Y -42.178,Z -194.684,A -90.000,B 90.000,C 0.000} C_DIS
LIN {X 11.237,Y -42.167,Z -194.411,A -90.000,B 90.000,C 0.000} C_DIS
LIN {X 12.087,Y -42.109,Z -192.946,A -90.000,B 90.000,C 0.000} C_DIS
LIN {X 13.183,Y -42.008,Z -191.077,A -90.000,B 90.000,C 0.000} C_DIS
LIN {X 13.280,Y -42.002,Z -190.923,A -90.000,B 90.000,C 0.000} C_DIS
LIN {X 13.828,Y -41.964,Z -190.112,A -90.000,B 90.000,C 0.000} C_DIS
LIN {X 14.200,Y -41.946,Z -189.558,A -90.000,B 90.000,C 0.000} C_DIS
LIN {X 15.558,Y -41.836,Z -187.357,A -90.000,B 90.000,C 0.000} C_DIS
LIN {X 15.662,Y -41.830,Z -187.199,A -90.000,B 90.000,C 0.000} C_DIS
LIN {X 15.833,Y -41.816,Z -186.949,A -90.000,B 90.000,C 0.000} C_DIS
LIN {X 15.876,Y -41.813,Z -186.889,A -90.000,B 90.000,C 0.000} C_DIS
LIN {X 16.596,Y -41.773,Z -185.926,A -90.000,B 90.000,C 0.000} C_DIS
LIN {X 17.058,Y -41.758,Z -185.302,A -90.000,B 90.000,C 0.000} C_DIS
LIN {X 18.023,Y -41.693,Z -183.889,A -90.000,B 90.000,C 0.000} C_DIS
LIN {X 18.110,Y -41.685,Z -183.764,A -90.000,B 90.000,C 0.000} C_DIS
LIN {X 18.258,Y -41.675,Z -183.565,A -90.000,B 90.000,C 0.000} C_DIS
LIN {X 19.199,Y -41.631,Z -182.397,A -90.000,B 90.000,C 0.000} C_DIS
LIN {X 19.808,Y -41.590,Z -181.653,A -90.000,B 90.000,C 0.000} C_DIS
LIN {X 20.628,Y -41.553,Z -180.711,A -90.000,B 90.000,C 0.000} C_DIS
LIN {X 21.325,Y -41.526,Z -179.935,A -90.000,B 90.000,C 0.000} C_DIS
LIN {X 22.579,Y -41.457,Z -178.554,A -90.000,B 90.000,C 0.000} C_DIS
LIN {X 22.844,Y -41.445,Z -178.262,A -90.000,B 90.000,C 0.000} C_DIS
LIN {X 22.995,Y -41.440,Z -178.102,A -90.000,B 90.000,C 0.000} C_DIS
LIN {X 23.790,Y -41.397,Z -177.217,A -90.000,B 90.000,C 0.000} C_DIS
LIN {X 24.168,Y -41.380,Z -176.805,A -90.000,B 90.000,C 0.000} C_DIS
LIN {X 24.445,Y -41.364,Z -176.506,A -90.000,B 90.000,C 0.000} C_DIS
LIN {X 24.849,Y -41.351,Z -176.060,A -90.000,B 90.000,C 0.000} C_DIS
LIN {X 25.604,Y -41.308,Z -175.184,A -90.000,B 90.000,C 0.000} C_DIS
LIN {X 25.604,Y -60.000,Z -175.184,A -90.000,B 90.000,C 0.000} C_DIS
LIN {X -21.348,Y -60.000,Z -215.201,A -90.000,B 90.000,C 0.000} C_DIS
LIN {X -21.348,Y -41.308,Z -215.201,A -90.000,B 90.000,C 0.000} C_DIS
LIN {X -21.149,Y -41.323,Z -215.134,A -90.000,B 90.000,C 0.000} C_DIS
LIN {X -20.662,Y -41.351,Z -214.973,A -90.000,B 90.000,C 0.000} C_DIS
LIN {X -19.905,Y -41.377,Z -214.679,A -90.000,B 90.000,C 0.000} C_DIS
LIN {X -18.767,Y -41.406,Z -214.222,A -90.000,B 90.000,C 0.000} C_DIS
LIN {X -18.520,Y -41.417,Z -214.134,A -90.000,B 90.000,C 0.000} C_DIS
LIN {X -18.186,Y -41.441,Z -214.025,A -90.000,B 90.000,C 0.000} C_DIS
LIN {X -17.972,Y -41.459,Z -213.964,A -90.000,B 90.000,C 0.000} C_DIS
LIN {X -17.546,Y -41.501,Z -213.858,A -90.000,B 90.000,C 0.000} C_DIS
LIN {X -15.968,Y -41.659,Z -213.472,A -90.000,B 90.000,C 0.000} C_DIS
LIN {X -13.921,Y -41.866,Z -212.918,A -90.000,B 90.000,C 0.000} C_DIS
LIN {X -13.680,Y -41.883,Z -212.836,A -90.000,B 90.000,C 0.000} C_DIS
LIN {X -13.634,Y -41.885,Z -212.821,A -90.000,B 90.000,C 0.000} C_DIS
LIN {X -12.990,Y -41.902,Z -212.576,A -90.000,B 90.000,C 0.000} C_DIS
LIN {X -12.616,Y -41.913,Z -212.439,A -90.000,B 90.000,C 0.000} C_DIS
LIN {X -11.801,Y -41.948,Z -212.140,A -90.000,B 90.000,C 0.000} C_DIS
LIN {X -11.685,Y -41.954,Z -212.102,A -90.000,B 90.000,C 0.000} C_DIS
LIN {X -11.393,Y -41.971,Z -212.015,A -90.000,B 90.000,C 0.000} C_DIS
LIN {X -11.089,Y -41.992,Z -211.936,A -90.000,B 90.000,C 0.000} C_DIS
LIN {X -10.820,Y -42.013,Z -211.880,A -90.000,B 90.000,C 0.000} C_DIS
LIN {X -10.475,Y -42.044,Z -211.821,A -90.000,B 90.000,C 0.000} C_DIS
LIN {X -10.236,Y -42.068,Z -211.790,A -90.000,B 90.000,C 0.000} C_DIS
LIN {X -9.794,Y -42.116,Z -211.746,A -90.000,B 90.000,C 0.000} C_DIS
LIN {X -9.216,Y -42.186,Z -211.687,A -90.000,B 90.000,C 0.000} C_DIS
LIN {X -7.770,Y -42.320,Z -211.378,A -90.000,B 90.000,C 0.000} C_DIS
LIN {X -7.463,Y -42.330,Z -211.246,A -90.000,B 90.000,C 0.000} C_DIS
LIN {X -7.298,Y -42.332,Z -211.179,A -90.000,B 90.000,C 0.000} C_DIS
LIN {X -7.095,Y -42.335,Z -211.110,A -90.000,B 90.000,C 0.000} C_DIS
LIN {X -6.819,Y -42.343,Z -211.023,A -90.000,B 90.000,C 0.000} C_DIS
